(* CoDeSys 2.3.9.50 project: Palettierer.pro *)
(* Libraries: TcIoFunctions.lib 20.1.15 18:06:58, TcXmlDataSrv.lib 11.7.11 07:38:08, STANDARD.LIB 5.6.98 13:03:02, TcBase.lib 14.5.09 13:14:08, TcEtherCAT.lib 9.1.15 17:08:56, TcMath.lib 23.9.04 16:15:30, TcSystem.lib 21.1.15 11:22:54, TcUtilities.lib 6.1.15 17:45:04, TcBaseMath.lib 27.7.04 13:07:56, TcTestAndSet.lib 23.2.09 13:50:08, TcpIp.lib 6.5.15 10:25:52, TcSocketHelper.lib 29.8.14 13:06:24, TcMDP.lib 5.12.13 13:01:38 *)

(* Global variable list: zLibrary/EsponRobot/gEpsonRobot *)
VAR_GLOBAL
	POS_PARK				: DINT := 1;
	POS_RT				: DINT := 21;
	POS_RT_WAIT			: DINT := 22;
	POS_WT_POS1		: DINT := 31;
	POS_WT_POS1_WAIT	: DINT := 32;
	POS_WT_POS2		: DINT := 35;
	POS_CAM_POS1		: DINT := 41;
	POS_CAM_POS2		: DINT := 45;
	POS_NOK				: DINT := 51;
	POS_FEED_PAL_WAIT 	: DINT := 100;
	POS_BUFFER_WAIT	: DINT := 100;
	POS_PAL_WAIT		: DINT := 200;
	POS_TEST_PARTS		: DINT := 300;
END_VAR

(* Global variable list: System/gGlobalSystem *)
VAR_GLOBAL
	Color 					: sColorCode;

	gReadyForControlOn		: BOOL;

	vGlbImpuls_1000ms		: BOOL;
	vGlbImpuls_0500ms		: BOOL;
	vGlbImpuls_0100ms		: BOOL;
	vGlbImpuls_0050ms		: BOOL;
	vGlbImpuls_0025ms		: BOOL;

(*Global Vars for Behr-System-Control *)
	gTipImp					: BOOL;
	gResetAll				: BOOL;
	gInitCollect				: BOOL;
	gInitOk					: BOOL;
	gSetupOk				: BOOL;
	gHomeOk				: BOOL;

(*SystemFlags for SFCs*)
	SFCInit					: BOOL:= FALSE;	(* Systemvariable for stop and reset an SFC *)
											(* Systemvariable zum stoppen und zurücksetzen einer Kette *)
	SFCQuitError			: BOOL:= FALSE;	(* Systemvariable for quitting an SFCError *)
											(* Systemvariable zum Quittieren des SFCErrors *)
	SFCError				: BOOL:= FALSE;	(* Systemvariable for checking Timeout in the step flow chart *)
											(* Systemvariable zur Anzeige eines Schrittkettentimeouts *)
	SFCErrorStep			: STRING:= '';	(* Systemvariable showing step of SFCError in step flow chart *)
											(* Systemvariable zur Anzeige des Schrittes in der der SFCError auftrat *)
	SFCErrorPOU			: STRING:= '';	(* Systemvariable showing Name of the  step flow chart, where SFCError occurs *)
											(* Systemvariable zur Anzeige des Namens der Schrittkette in der der SFCError auftrat *)
	SFCTip  				: BOOL:= FALSE;	(* Systemvariable zum forcen aller Transitionen auf TRUE (! DO NOT USE !) *)
											(* Systemvariable to force all Transitions*)
	SFCTipMode			: BOOL:= FALSE;	(* Systemvariable zum anhalten der AS-Diagramme an den Transitionen *)
											(* Systemvariable to stop an AS-Diagram at the transition *)
	gVarStrSystemTime 		: STRING;
	gVarDTSystemtime		: DT;
	gVarSystemtime			: TIMESTRUCT;

	LocalAmsNetIdArr		: T_AmsNetIdArr;
	LocalAmsNetIdStr		: T_AmsNetId;
	Analyze					: AnalyzeExpression;

	st_Hydra8Data			: struct_Hydra8;
	FbExportHydraString		: Fb_ExportHydraString;

	st_ctrl_in_Empty		: struct_ctrl_in;
	st_ctrl_out_Empty		: struct_ctrl_out;

END_VAR
VAR_GLOBAL CONSTANT
	NO_OF_POS_AXIS		: INT :=3;
	NO_OF_ERRORS		: DINT :=30;
	NO_OF_USERS			: DINT :=50;
	NO_OF_FILES			: DINT :=50;
END_VAR

(* Global variable list: System/gGlobalVisuPersist *)
VAR_GLOBAL
	Visu		 AT %MB1000 : sVisu;
	Service		: sMachParaService;
END_VAR

VAR_GLOBAL RETAIN PERSISTENT
	TD			: sTypeData;
	MP			: sMachPara;
	UD			: sUserList;


	sTDHandler 	: sTDHandler;
	sMPHandler 	: sMPHandler;
	ErrorHistory	: ARRAY[0..500] OF ErrorStruct;

	lastTDActivate	: STRING(255);

	(*Gesamt-Zähler (Reset möglich durch Service*)
	gNOKCount			: DINT;

	(*Gesamt-Zähler (Reset nur möglich durch Administrator*)
	gTotalNOKCount		: DINT;


	PersDaten			: sPersDaten;

END_VAR

(* Global variable list: ept/Global_Checks *)
VAR_GLOBAL
	CheckBounds_ErrCnt 			: DINT := 0;
	CheckByteZeroDiv_ErrCnt 		: DINT := 0;
	CheckDWordZeroDiv_ErrCnt 	: DINT := 0;
	CheckRealZeroDiv_ErrCnt 		: DINT := 0;
	CheckWordZeroDiv_ErrCnt 		: DINT := 0;
	CheckRangeSigned_ErrCnt		: DINT := 0;
	CheckRangeUnsigned_ErrCnt	: DINT := 0;
END_VAR

(* Global variable list: zLibrary/Valve/gValve *)
 VAR_GLOBAL
	gValve		:	sValveGlobalVar;
END_VAR

(* Global variable list: System/MachineParameterFix *)
VAR_GLOBAL

	MP_TDPathLocal			: STRING(255) := 'data\TD\';
	MP_TDPathService		: STRING(255):= 'data\TD\Service\';

	MP_LocalDriveRoot		: STRING(255) := 'data\MP\';

	MP_ExportDrive			: STRING:=	'';

	MP_ExportDrivePathTD	: STRING(255):=  'data\TD';
	MP_ExportDrivePathMP	: STRING(255):=  'data\MP';

	LOG_RDPathLocal			: STRING(255) := 'data\RD\';
	LOG_ExportDrivePathRD	: STRING(255):= 'data\RD';

	MP_TDFileExtension		: STRING(10) := '.XML';
	MP_TDSearchString		: STRING :=  '*.xml';
	MP_MPExportFilename		: STRING := 'MachPara.xml';

	s_PLC_name				: STRING(255);
	s_PLC_path				: STRING(255);
	s_Projekt_path			: STRING(255);

	s_tools_path			: STRING(255):= 'tools\';
	s_ud_path				: STRING(255):= 'data\UD\';

END_VAR

(* Global variable list: Station00/ST00_FBs *)
VAR_GLOBAL
	ST00_40_F1 			: FB_DigIn; (* Vorsicherungen Leistung iO *)
	ST03_210_S1 			: FB_DigIn; (* Not-Aus 1 Anlage ausgelöst *)
	ST08_210_S2 			: FB_DigIn; (* Not-Aus 2 Anlage ausgelöst *)
	ST00_X4_16	 		: FB_DigIn; (* Not-Aus Reserve Anlage ausgelöst *) (*entfällt*)
	ST00_200_A1_A1 		: FB_DigIn; (* Not-Aus iO *)
	ST00_220_S1	 		: FB_DigIn; (* Schutztüre 1 geöffnet *)
	ST00_220_S2			: FB_DigIn; (* Schutztüre 2 geöffnet *)
	ST00_230_S2_E1 		: FB_DigIn; (* Schutztüre 1 geschlossen *)
	ST00_240_S1 			: FB_DigIn; (* Schutztüre 9 geschlossen *)
	ST00_226_S1			: FB_DigIn;(*Hubtüre 1 Schleuse Einlauf STN 8 geschlossen*)
	ST00_226_S2			: FB_DigIn;(*Hubtüre 2 Schleuse Einlauf STN 8 geschlossen*)
	ST00_227_S1			: FB_DigIn;(*Hubtüre 3 Schleuse Auslauf STN 8 geschlossen*)
	ST00_227_S2			: FB_DigIn;(*Hubtüre 4 Schleuse Auslauf STN 8 geschlossen*)
	ST00_229_S1			: FB_DigIn;(*Schutztüre Einlauf Tray STN 8 geschlossen*)
	ST00_230_S1			: FB_DigIn;(*Schutztüre Auslauf Tray STN 8 geschlossen*)
	ST00_231_S1			: FB_DigIn;(*Schutztüre Panel / Rutsche STN 8 geschlossen*)
	ST00_232_S1			: FB_DigIn;(*Schutztüre 8 Auslauf Trays STN 8 geschlossen*)
	ST00_170_Motorschutz	: FB_DigIn;(*Motorschutz in Ordnung*)
	ST00_170_Thermokont	: FB_DigIn;(*Thermokontakt in Ordnung*)
	ST00_228_S1			: FB_DigIn;(*Bandstecke EPT angebaut*)
	ST00_71_X1_3  		: FB_DigIn; (* Schnittstelle Bedrucken Tinte JSK auf Übergabeposition *)
	ST00_71_X1_4  		: FB_DigIn; (* Schnittstelle Bedrucken Tinte Druckstation betriebsbereit *)
	ST00_72_X1_3  		: FB_DigIn; (* Schnittstelle Tampondrucker Teil in Abholposition *)(*Band Entnahmeposition 1*)
	ST00_72_X1_8  		: FB_DigIn; (* Schnittstelle Tampondrucker Druck abgeschlossen *)	(*gleich wie ST02_S2_B11_0*)
	ST00_292_S1_STOP 	: FB_DigIn; (* Bedienstelle Produktion Stop *)
	ST00_292_S2_START	: FB_DigIn; (* Bedienstelle Produktion Start *)
	ST00_292_S3_RESET	: FB_DigIn; (* Bedienstelle Produktion Reset *)
	ST00_350_B20_0 		: FB_DigIn; (* Druckschalter Wartungseinheit Hauptluft min.6 bar *)

	ST00_245_V1			: FB_DigOutIn; (* Verriegelung Schutztüren-Leuchte *)
	ST00_245_V2_START	: FB_DigOutIn; (* Bedienstelle Start-Leuchte *)
	ST00_245_V3_RESET	: FB_DigOutIn; (* Bedienstelle Reset-Schutztüren-Leuchte *)
	ST00_245_S1_STOP 	: FB_DigIn;	(* Bedienstelle Produktion Stop *)
	ST00_245_S2_START	: FB_DigIn; (* Bedienstelle Produktion Start *)
	ST00_245_S3_RESET	: FB_DigIn; (* Bedienstelle Produktion Reset *)

	ST00_31_K1 			: FB_DigOutIn; (* Beleuchtung Anlage *)
	ST00_350_H1			: FB_DigOutIn; (* Signalsäule RD Maschine Alarm/Störung *)
	ST00_350_H2			: FB_DigOutIn; (* Signalsäule YE Bedienereingriff erforderlich *)
	ST00_350_H3			: FB_DigOutIn; (* Signalsäule GN Maschine Automatik *)
	ST00_200_A1_E4 		: FB_DigOutIn; (* Quittierung Not-Aus *)
	ST00_220_S1_S31		: FB_DigOutIn; (* Verriegelung Schutztüren *)
	ST00_292_H2_START	: FB_DigOutIn; (* Bedienstelle Start-Leuchte *)
	ST00_292_H3_RESET	: FB_DigOutIn; (* Bedienstelle Reset-Leuchte *)

	ST00_71_K2	  		: FB_DigOutIn; (* Schnittstelle Bedrucken Tinte Abholposition frei *)
	ST00_72_K7	  		: FB_DigOutIn; (* Schnittstelle Tampondrucker Reset  Rundtisch *)

	ST00_73_K3	  		: FB_DigOutIn; (* Schnittstelle Förderband frei für Spritzmaschine*)
	ST00_73_K4	  		: FB_DigIn; 		(* Schnittstelle Freigabe von Spritzmaschine (nur für Anlagen ohne Rundtisch)*)
	ST00_74_B7_2    		: FB_ValveSensor; (* Stopper GST1 DS*)
	ST00_74_B7_3   		: FB_ValveSensor; (* Stopper GST2 PS*)
	ST00_74_B7_4    		: FB_ValveSensor; (* Vereinzeler AST1 DS*)
	ST00_74_B7_5   	 	: FB_ValveSensor; (* Vereinzeler AST2 PS*)
	ST00_74_B7_6  	 	: FB_ValveSensor; (* Vereinzeler GST1 DS*)
	ST00_74_B7_7   		: FB_ValveSensor; (* Vereinzeler GST2 PS*)

	ST00_74_Y2_4    		: FB_Valve; (*ST00_74_Y2_4 Stopper Bandstrecke (Valve) *)
	ST00_74_Y2_5    		: FB_Valve; (*ST00_74_Y2_5 Vereinzeler Bandstrecke (Valve) *)

END_VAR

(* Global variable list: Station00/ST00_Global *)
VAR_GLOBAL
	gDisableMP				: BOOL := FALSE;		(* deaktivieren der Maschinenparamtereingabe *)
	gDisableTD				: BOOL := FALSE;		(* deaktivieren der Typedateneingabe *)

	gHomePosSFCDone		: BOOL;
	gResetButton		: BOOL;
	gRobotOffset		: DINT;
	gTypeCode		  	: DINT;
	ProcessMessage01	: STRING(80);
	ProcessMessage02	: STRING(80);
	gTInfo_FirstStart	: BOOL;
	gBasicManualMode	: BOOL;
	SpecialModeProgNu	: DINT;

	gStartRunEmpty		: BOOL;
	gRunEmpty			: BOOL;

	DummyTest_160pol	: BOOL;
	Dummy_test_Result	: ARRAY[1..MAX_NO_OF_DUMMYS] OF BOOL;
	Dummy_test_Vorgabe	: ARRAY[1..MAX_NO_OF_DUMMYS] OF BOOL;

END_VAR
VAR_GLOBAL RETAIN PERSISTENT
	gTypeDataValid		 : BOOL;
END_VAR
VAR_GLOBAL CONSTANT
	MAX_NO_OF_DUMMYS	: DINT := 6;
END_VAR

(* Global variable list: Station00/ST00_VarVonfig *)
VAR_CONFIG
	BusDiagnosis.EtheCatMasterAmsNetId AT %IB1000 : ARRAY [0..5] OF USINT;

(* Vorsicherungen Leistung iO *)
.ST00_40_F1.BitInToCheck                 	AT %IX0.0 : BOOL;
(* Schutztüre 2 geöffnet *)
.ST00_220_S2.BitInToCheck                 AT %IX0.2 : BOOL;
(* Not-Aus 1 Anlage ausgelöst *)
.ST03_210_S1.BitInToCheck                 AT %IX0.3 : BOOL;
(* Not-Aus 2 Anlage ausgelöst *)
.ST08_210_S2.BitInToCheck                 AT %IX0.4 : BOOL;
(* Not-Aus Reserve Anlage ausgelöst *)
.ST00_X4_16.BitInToCheck                 	AT %IX0.5 : BOOL;
(* Not-Aus iO *)
.ST00_200_A1_A1.BitInToCheck              AT %IX0.6 : BOOL;
(* Schutztüre 9 geschlossen *)
.ST00_240_S1.BitInToCheck                 AT %IX0.7 : BOOL;
(* Schutztüre 1 geöffnet *)
.ST00_220_S1.BitInToCheck                 AT %IX1.0 : BOOL;
(* Schutztüre 1 geschlossen *)
.ST00_230_S2_E1.BitInToCheck              AT %IX1.1 : BOOL;
(*Hubtüre 1 Schleuse Einlauf STN 8 geschlossen*)
.ST00_226_S1.BitInToCheck                 AT %IX1.2 : BOOL;
(*Hubtüre 2 Schleuse Einlauf STN 8 geschlossen*)
.ST00_226_S2.BitInToCheck                 AT %IX1.3 : BOOL;
(*Hubtüre 3 Schleuse Auslauf STN 8 geschlossen*)
.ST00_227_S1.BitInToCheck                 AT %IX1.4 : BOOL;
(*Hubtüre 4 Schleuse Auslauf STN 8 geschlossen*)
.ST00_227_S2.BitInToCheck                 AT %IX1.5 : BOOL;
(*Motorschutz in Ordnung*)
	ST00_170_Motorschutz.BitInToCheck	AT %IX1.6 : BOOL;
(*Thermokontakt in Ordnung*)
	ST00_170_Thermokont.BitInToCheck	AT %IX1.7 : BOOL;

(* Schnittstelle Bedrucken Tinte JSK auf Übergabeposition *)
.ST00_71_X1_3.BitInToCheck                AT %IX2.0 : BOOL;
(* Schnittstelle Bedrucken Tinte Druckstation betriebsbereit *)
.ST00_71_X1_4.BitInToCheck                AT %IX2.1 : BOOL;
(* Schnittstelle Tampondrucker Teil in Abholposition *)
.ST00_72_X1_3.BitInToCheck                AT %IX2.2 : BOOL;

(* Schnittstelle Tampondrucker Druck abgeschlossen *)
.ST00_72_X1_8.BitInToCheck                AT %IX2.7 : BOOL;
(*Bandstecke EPT angebaut*)
.ST00_228_S1.BitInToCheck                 AT %IX3.0 : BOOL;

(*Schutztüre Einlauf Tray STN 8 geschlossen*)
.ST00_229_S1.BitInToCheck                 AT %IX3.2 : BOOL;
(*Schutztüre Auslauf Tray STN 8 geschlossen*)
.ST00_230_S1.BitInToCheck                 AT %IX3.3 : BOOL;
(*Schutztüre Panel / Rutsche STN 8 geschlossen*)
.ST00_231_S1.BitInToCheck                 AT %IX13.0 : BOOL;
(*Schutztüre 8 Auslauf Trays STN 8 geschlossen*)
.ST00_232_S1.BitInToCheck                 AT %IX13.1 : BOOL;

(* Bedienstelle Produktion Stop *)
.ST00_292_S1_STOP.BitInToCheck            AT %IX3.5 : BOOL;
(* Bedienstelle Produktion Start *)
.ST00_292_S2_START.BitInToCheck           AT %IX3.6 : BOOL;
(* Bedienstelle Produktion Start *)
.ST00_292_S3_RESET.BitInToCheck           AT %IX3.7 : BOOL;
(* Druckschalter Wartungseinheit Hauptluft min.6 bar *)
.ST00_350_B20_0.BitInToCheck           		AT %IX20.0 : BOOL;

(* Beleuchtung Anlage *)
.ST00_31_K1.BitInToCheck             		: BOOL := FALSE;
.ST00_31_K1.BitOutToSet              		  AT %QX0.0 : BOOL;
(* Signalsäule RD Maschine Alarm/Störung *)
.ST00_350_H1.BitInToCheck             	: BOOL := FALSE;
.ST00_350_H1.BitOutToSet              	  AT %QX0.4 : BOOL;
(* Signalsäule YE Bedienereingriff erforderlich *)
.ST00_350_H2.BitInToCheck             	: BOOL := FALSE;
.ST00_350_H2.BitOutToSet              	  AT %QX0.5 : BOOL;
(* Signalsäule GN Maschine Automatik *)
.ST00_350_H3.BitInToCheck             	: BOOL := FALSE;
.ST00_350_H3.BitOutToSet              	  AT %QX0.6 : BOOL;
(* Quittierung Not-Aus *)
.ST00_200_A1_E4.BitInToCheck            : BOOL := FALSE;
.ST00_200_A1_E4.BitOutToSet               AT %QX1.0 : BOOL;
(* Verriegelung Schutztüren *)
.ST00_220_S1_S31.BitInToCheck           : BOOL := FALSE;
.ST00_220_S1_S31.BitOutToSet              AT %QX1.1 : BOOL;
(* Bedienstelle Start-Leuchte *)
.ST00_292_H2_START.BitInToCheck         : BOOL := FALSE;
.ST00_292_H2_START.BitOutToSet            AT %QX1.5 : BOOL;
(* Bedienstelle Reset-Leuchte *)
.ST00_292_H3_RESET.BitInToCheck         : BOOL := FALSE;
.ST00_292_H3_RESET.BitOutToSet            AT %QX1.7 : BOOL;

(* Schnittstelle Bedrucken Tinte Abholposition frei *)
.ST00_71_K2.BitInToCheck             		: BOOL := FALSE;
.ST00_71_K2.BitOutToSet              		  AT %QX2.1 : BOOL;

(* Schnittstelle Förderband frei für Spritzmaschine*)
.ST00_73_K3.BitInToCheck             		: BOOL := FALSE;
.ST00_73_K3.BitOutToSet              		  AT %QX0.7 : BOOL;


(*ST00_74_Y2_4 Stopper Bandstrecke (Valve) *)
.ST00_74_Y2_4.CoilA                    AT %QX2.4 : BOOL;
.ST00_74_Y2_4.CoilB                    AT %MX2.4 : BOOL;

(*ST00_74_Y2_5 Vereinzeler Bandstrecke (Valve) *)
.ST00_74_Y2_5.CoilA                    AT %QX2.5 : BOOL;
.ST00_74_Y2_5.CoilB                    AT %MX2.5 : BOOL;

(*ST00_74_B7_2 Stopper GST1 DS (DigIn) *)
.ST00_74_B7_2.ValveSensor             AT %IX7.2 : BOOL;

(*ST00_74_B7_3 Stopper GST2 PS (DigIn) *)
.ST00_74_B7_3.ValveSensor             AT %IX7.3 : BOOL;

(*ST00_74_B7_4 Vereinzeler AST1 DS (DigIn) *)
.ST00_74_B7_4.ValveSensor             AT %IX7.4 : BOOL;

(*ST00_74_B7_5 Vereinzeler AST2 PS (DigIn) *)
.ST00_74_B7_5.ValveSensor             AT %IX7.5 : BOOL;

(*ST00_74_B7_6 Vereinzeler GST1 DS (DigIn) *)
.ST00_74_B7_6.ValveSensor          AT %IX7.6: BOOL;

(*ST00_74_B7_7 Vereinzeler GST2 PS(DigIn) *)
.ST00_74_B7_7.ValveSensor             AT %IX7.7 : BOOL;


END_VAR

(* Global variable list: Station02/ST02_FBs *)
VAR_GLOBAL
	ST02_FDB_55X1_5_READY		:FB_DigIn; (* IFM Kamera Flügelerkennung links Ready *)
	ST02_FDB_55X1_6_IO			 :FB_DigIn; (* IFM Kamera Flügelerkennung links Ergebnis iO *)
	ST02_FDB_55X1_6_NIO		:FB_DigIn; (* IFM Kamera Flügelerkennung links Ergebnis niO *)
	ST02_FDB_55X1_2_TRIGGER	:FB_DigOutIn; (* IFM Kamera Flügelerkennung links Trigger *)
	ST02_FDB_55X1_7_JOB_BIT1 	:FB_DigOutIn; (* IFM Kamera links  Jobwechsel Bit 1 *)
	ST02_FDB_55X1_7_JOB_BIT2 	:FB_DigOutIn; (* IFM Kamera links Jobwechsel Bit 2 *)

	ST02_FDB_56X1_5_READY		:FB_DigIn; (* IFM Kamera Flügelerkennung rechts Ready *)
	ST02_FDB_56X1_6_IO			:FB_DigIn; (* IFM Kamera Flügelerkennung rechts Ergebnis iO *)
	ST02_FDB_56X1_6_NIO		:FB_DigIn; (* IFM Kamera Flügelerkennung rechts Ergebnis niO *)
	ST02_FDB_56X1_2_TRIGGER	:FB_DigOutIn; (* IFM Kamera Flügelerkennung rechts Trigger *)
	ST02_FDB_56X1_7_JOB_BIT1	:FB_DigOutIn; (* IFM Kamera links  Jobwechsel Bit 1 *)
	ST02_FDB_56X1_7_JOB_BIT2	:FB_DigOutIn; (* IFM Kamera links Jobwechsel Bit 2 *)


	ST02_DT_95_A1 			:FB_Sensopart;	(*Sensopart Kamera Farberkennung*)
	ST02_DT_95_A2 			:FB_SensopartEthernet;	(*Sensopart Kamera Farberkennung*)

	ST02_S1_70K61_A1		:FB_DigOutIn; 	(* Start  Bedrucken *)

	ST02_DT_62_B11		:FB_ValveSensor;	(* Schwenkarm 1 0 Grad*)
	ST02_DT_61_B21		:FB_ValveSensor;	(* Schwenkarm 2 90 Grad*)
	ST02_DT_61_B11		:FB_ValveSensor;	(* Schwenkarm 2 180 Grad*)
	ST02_DT_61_B31		:FB_ValveSensor;	(* Schwenkarm 2 0 Grad*)
	ST02_DT_61_B41 		:FB_ValveSensor;	(* Schwenkarm 1 180 Grad*)
	ST02_DT_61_B51 		:FB_ValveSensor;	(* Schwenkarm 1 90 Grad*)
	ST02_FDB_54_B11		:FB_ValveSensor; 	(* Kamera Ausschleusen Bandstrecke eingefahren GST*)
	ST02_FDB_54_B21		:FB_ValveSensor; 	(* Kamera Ausschleusen Bandstrecke ausgefahren AST*)
	ST02_S1_66_B11 		:FB_ValveSensor;	(*9: Schwenkarm 1 ISK Fixierung GST*)
	ST02_S1_66_B21 		:FB_ValveSensor;	(*10: Schwenkarm 1 ISK Fixierung AST*)
	ST02_S1_66_B31 		:FB_ValveSensor;	(*11: Schwenkarm 2 ISK Fixierung GST*)
	ST02_S1_66_B41	 	:FB_ValveSensor;	(*12: Schwenkarm 2 ISK Fixierung AST*)

	ST02_FDB_40_B61		:FB_DigIn; (* Iso von SPM auf Band abgelegt *)
	ST02_FDB_40_B71		:FB_DigIn; (* Iso auf Band vor Vereinzler *)

	ST02_DT_62_B81		:FB_ValveSensor; 	(* Tisch drehen 0 Grad*)			(*gleich wie ST00_72_X1_6*)
	ST02_DT_62_B91		:FB_ValveSensor;	(* Tisch drehen 180 Grad*)			(*gleich wie ST00_72_X1_7*)
	ST02_S1_40K01 		:FB_DigIn;			(* Freigabe Förderband von SPM*)

	ST02_FDB_80_B02 		:FB_DigIn;			(* Band Entnahmeposition 2 102pol*)
	ST02_FDB_54_B41		:FB_DigIn; 			(* Kamera ISK anwesend an Prüfposition nur zum Schlechtteile zählen*)
	ST02_35_S31 			:FB_DigIn; 			(* ST02 Druckschalter Wartungseinheit Hauptluft min.6 bar *)
	ST02_S1_6A01			:FB_DigIn; 			(* ST02 Sicherung 24V *)

	ST02_35Y01			:FB_Valve; 			(*1: Einschaltventil Hauptluft Tampondruckanlage*)

	ST02_62_Y4  			:FB_Valve; 			(*Kamera Ausschleusen Bandstrecke (Valve) *)
	ST02_62_Y6			:FB_Valve; 			(*Tisch drehen 0 - 180 Grad (Valve) *)

	ST02_Schwenkarm	: ARRAY[1..2] OF FB_Schwenken;
	ST02_62_Y9			:FB_Valve; 			(*Schwenkarm 2 drehen 90 - 180 Grad (Valve) *)
	ST02_62_Y11			:FB_Valve; 			(*Schwenkarm 2 drehen 90 - 0 Grad (Valve) *)

	ST02_62_Y13			:FB_Valve; 			(*Schwenkarm 1 drehen 90 - 180 Grad (Valve) *)
	ST02_62_Y15			:FB_Valve; 			(*Schwenkarm 1 drehen 90 - 0 Grad (Valve) *)

	ST02_62_Y17			:FB_Valve; 			(*Schwenkarm 1 ISK Fixierung ein/ausfahren(Valve)*)
	ST02_62_Y18			:FB_Valve; 			(*Schwenkarm 2 ISK Fixierung ein/ausfahren(Valve)*)

	ST02_DT_65B11  		:FB_DigIn;			(* Tampondrucker Nest 1 leer *)
	ST02_DT_65B21		:FB_DigIn; 			(* Tampondrucker Nest 2 leer *)

END_VAR

(* Global variable list: Station02/ST02_Global *)
VAR_GLOBAL
	gTableEmpty			: BOOL;
END_VAR

VAR_GLOBAL CONSTANT
	NO_OF_NEST			: INT := 2;		(* No of Nests on TurnTable *)
END_VAR

(* Global variable list: Station02/ST02_VarVonfig *)
(* Generated automatically by TwinCAT - (read only) *)
VAR_CONFIG

(*ST02_FDB_55X1_5_READY IFM Kamera Flügelerkennung links Ready (DigIn) *)
.ST02_FDB_55X1_5_READY.BitInToCheck           AT %IX100.1 : BOOL;
(*ST02_FDB_55X1_6_IO IFM Kamera Flügelerkennung links Ergebnis iO (DigIn) *)
.ST02_FDB_55X1_6_IO.BitInToCheck         		  AT %IX100.2 : BOOL;
(*ST02_FDB_55X1_6_NIO IFM Kamera Flügelerkennung links Ergebnis niO (DigIn) *)
.ST02_FDB_55X1_6_NIO.BitInToCheck        		   AT %IX100.3 : BOOL;
(*ST02_FDB_55X1_2_TRIGGER IFM Kamera Flügelerkennung links Trigger (DigOutIn) *)
.ST02_FDB_55X1_2_TRIGGER.BitInToCheck                : BOOL := FALSE;
.ST02_FDB_55X1_2_TRIGGER.BitOutToSet                 AT %QX100.1 : BOOL;
(* IFM Kamera links  Jobwechsel Bit 1 *)
.ST02_FDB_55X1_7_JOB_BIT1.BitInToCheck                : BOOL := FALSE;
.ST02_FDB_55X1_7_JOB_BIT1.BitOutToSet                 AT %QX100.2 : BOOL;
(* IFM Kamera links Jobwechsel Bit 2 *)
.ST02_FDB_55X1_7_JOB_BIT2.BitInToCheck                : BOOL := FALSE;
.ST02_FDB_55X1_7_JOB_BIT2.BitOutToSet                 AT %QX100.3 : BOOL;

(*ST02_FDB_56X1_5_READY IFM Kamera Flügelerkennung rechts Ready (DigIn) *)
.ST02_FDB_56X1_5_READY.BitInToCheck           AT %IX101.4 : BOOL;
(*ST02_FDB_56X1_6_IO IFM Kamera Flügelerkennung rechts Ergebnis iO (DigIn) *)
.ST02_FDB_56X1_6_IO.BitInToCheck           AT %IX101.5 : BOOL;
(*ST02_FDB_56X1_6_NIO IFM Kamera Flügelerkennung rechts Ergebnis niO (DigIn) *)
.ST02_FDB_56X1_6_NIO.BitInToCheck           AT %IX101.6 : BOOL;
(*ST02_FDB_56X1_2_TRIGGER IFM Kamera Flügelerkennung rechts Trigger (DigOutIn) *)
.ST02_FDB_56X1_2_TRIGGER.BitInToCheck                : BOOL := FALSE;
.ST02_FDB_56X1_2_TRIGGER.BitOutToSet                 AT %QX101.2 : BOOL;
(* IFM Kamera rechts  Jobwechsel Bit 1 *)
.ST02_FDB_56X1_7_JOB_BIT1.BitInToCheck                : BOOL := FALSE;
.ST02_FDB_56X1_7_JOB_BIT1.BitOutToSet                 AT %QX101.3 : BOOL;
(* IFM Kamera rechts Jobwechsel Bit 2 *)
.ST02_FDB_56X1_7_JOB_BIT2.BitInToCheck                : BOOL := FALSE;
.ST02_FDB_56X1_7_JOB_BIT2.BitOutToSet                 AT %QX101.4 : BOOL;


(*ST02_S1_70K61_A1 Start  Bedrucken (DigOutIn) *)
.ST02_S1_70K61_A1.BitInToCheck                : BOOL := FALSE;
.ST02_S1_70K61_A1.BitOutToSet                 AT %QX6.3: BOOL;

(*ST02_S1_40K01 Freigabe Förderband von SPM (DigIn)*)
.ST02_S1_40K01.BitInToCheck    AT %IX11.2 : BOOL;
(*ST02_FDB_80_B02  Band Entnahmeposition 2(DigIn) *)
.ST02_FDB_80_B02.BitInToCheck    AT %IX11.6 : BOOL;

(* Tampondrucker Nest 1 leer *)
.ST02_DT_65B11.BitInToCheck                AT %IX2.3 : BOOL;
(* Tampondrucker Nest 2 leer *)
.ST02_DT_65B21.BitInToCheck                AT %IX2.4 : BOOL;

(*ST02_DT_62_B11 Schwenkarm 1 0 Grad (DigIn) *)
.ST02_DT_62_B11.ValveSensor             AT %IX10.0 : BOOL;
(*ST02_DT_61_B21 Schwenkarm 2 90 Grad(DigIn) *)
.ST02_DT_61_B21.ValveSensor             AT %IX10.1 : BOOL;
(*ST02_DT_61_B11 Schwenkarm 2 180 Grad(DigIn) *)
.ST02_DT_61_B11.ValveSensor             AT %IX10.2 : BOOL;
(*ST02_DT_61_B31 Schwenkarm 2 0 Grad(DigIn) *)
.ST02_DT_61_B31.ValveSensor             AT %IX10.3 : BOOL;
(*ST02_DT_61_B41 Schwenkarm 1 180 Grad(DigIn) *)
.ST02_DT_61_B41.ValveSensor             AT %IX10.4 : BOOL;
(*ST02_DT_61_B51 Schwenkarm 1 90 Grad(DigIn) *)
.ST02_DT_61_B51.ValveSensor             AT %IX10.5 : BOOL;
(*ST02_DT_62_B81 Tisch drehen 0 Grad(DigIn) *)
.ST02_DT_62_B81.ValveSensor             AT %IX10.6 : BOOL;
(*ST02_DT_62_B91 Tisch drehen 180 Grad(DigIn) *)
.ST02_DT_62_B91.ValveSensor             AT %IX10.7 : BOOL;
(*
(*ST02_S1_66_B11 Schwenkarm 1 ISK Fixierung GST(DigIn) *)
.ST02_S1_66_B11.ValveSensor             AT %I* : BOOL;
(*ST02_S1_66_B21 Schwenkarm 1 ISK Fixierung AST(DigIn) *)
.ST02_S1_66_B21.ValveSensor             AT %I* : BOOL;
(*ST02_S1_66_B31 Schwenkarm 2 ISK Fixierung GST(DigIn) *)
.ST02_S1_66_B31.ValveSensor             AT %I* : BOOL;
(*ST02_S1_66_B41 Schwenkarm 2 ISK Fixierung AST(DigIn) *)
.ST02_S1_66_B41.ValveSensor             AT %I* : BOOL;

(* ST02 Druckschalter Wartungseinheit Hauptluft min.6 bar *)
.ST02_35_S31.BitInToCheck             AT %I* : BOOL;
(* ST02 Sicherung 24V *)
.ST02_S1_6A01.BitInToCheck             AT %I* : BOOL;
*)
(*
(*ST02_62V9a Schwenkarm 1 ISK Fixierung ein/ausfahren(Valve) (Valve) *)
.ST02_62V9a.CoilA                    AT %Q* : BOOL;
(*ST02_62V9b Schwenkarm 2 ISK Fixierung ein/ausfahren(Valve)  (Valve) *)
.ST02_62V9b.CoilB                    AT %Q* : BOOL;
*)
(*
(*ST02_62_Y6 Tisch drehen 0 - 180 Grad  (Valve) *)
.ST02_62_Y6.CoilA                    AT %QX5.6 : BOOL;
.ST02_62_Y6.CoilB                    AT %MX5.6 : BOOL;
(*ST02_62_Y9 Schwenkarm 2 drehen 90 - 180 Grad  (Valve) *)
.ST02_62_Y9.CoilA                    AT %QX5.7 : BOOL;
.ST02_62_Y9.CoilB                    AT %MX5.7 : BOOL;
(*ST02_62_Y11 Schwenkarm 2 drehen 90 - 0 Grad  (Valve) *)
.ST02_62_Y11.CoilA                    AT %QX6.0 : BOOL;
.ST02_62_Y11.CoilB                    AT %MX6.0 : BOOL;
(*ST02_62_Y13 Schwenkarm 1 drehen 90 - 180 Grad  (Valve) *)
.ST02_62_Y13.CoilA                    AT %QX6.1 : BOOL;
.ST02_62_Y13.CoilB                    AT %MX6.1 : BOOL;
(*ST02_62_Y15 Schwenkarm 1 drehen 90 - 0 Grad  (Valve) *)
.ST02_62_Y15.CoilA                    AT %QX6.2 : BOOL;
.ST02_62_Y15.CoilB                    AT %MX6.2 : BOOL;
*)
(*ST02_62_Y4 Kamera Ausschleusen Bandstrecke (Valve) *)
.ST02_62_Y4.CoilA                    AT %QX60.0 : BOOL;
.ST02_62_Y4.CoilB                    AT %QX60.1 : BOOL;

(*ST02_FDB_54_B11 Kamera Ausschleusen Bandstrecke eingefahren (DigIn) *)
.ST02_FDB_54_B11.ValveSensor             AT %IX60.0 : BOOL;
(*ST02_FDB_54_B21 Kamera Ausschleusen Bandstrecke ausgefahren (DigIn) *)
.ST02_FDB_54_B21.ValveSensor             AT %IX60.1 : BOOL;

(*ST02_FDB_54_B41 Kamera ISK anwesend an Prüfposition (DigIn) *)
.ST02_FDB_54_B41.BitInToCheck           AT %IX70.6 : BOOL;
(*
(*ST02_35Y01 Einschaltventil Hauptluft Tampondruckanlage (Valve) *)
.ST02_35Y01.CoilA                    AT %Q* : BOOL;
.ST02_35Y01.CoilB                    AT %Q* : BOOL;*)
END_VAR

(* Global variable list: Station03/ST03_FBs *)
VAR_GLOBAL

	ST03_51_M1	: fb_72x1_Achse;	(* Förderbandmotor*)
	ST03_601V1_A1: FB_DigOutIn;		(* Förderband Prüfteile *)
	ST03_A5		: FB_DigOutIn;		(* Förderbandmotor Oriental *)
	ST03_V2	 	: FB_DigIn; 		(* Störung Motor Förderband Oriental *)

	ST03_125_F1 : FB_DigIn; 		(* Absicherung Roboter iO *)
	Robot01		: FB_EpsonRobot;

	St03_120_A1_A14: FB_DigIn;		(* Roboter opt.- Tool 2 ist ein*)
	ST03_400_B12_6 : FB_DigIn; 		(* Schwenkmodul AST (Roboterkopf) *)
	ST03_400_B12_7 : FB_DigIn; 		(* Schwenkmodul GST (Roboterkopf) *)
	ST03_400_B54_7: FB_DigIn; 		(* Tray Testteile in Position *)
	ST03_8_75_B13_5: FB_DigIn; 		(* voll/belegt keine Prüfmittel mehr*)
	ST03_8_75_B13_6: FB_DigIn; 		(* belegt mit 6 Prüfmitteln*)

	ST03_BG3_S53_0:FB_DigIn;		(* Start Band für Dummyprüfung*)
	ST03_BG3_X53_0:	FB_DigOutIn;	(* LED TasterStart Band für Dummyprüfung*)

	ST03_65_Q1: FB_DigOutIn;		(* Kühltunnel (Lüfter)*)
	ST03_65_F1: FB_DigIn;			(* Sicherung Kühltunnel (Lüfter)*)

	ST03_8_100_A1	: FB_SensopartEthernet;	(*Sensopart Kamera Farberkennung*)
	ST03_8_103_A1	: FB_SensopartEthernet;	(*Sensopart Kamera Farberkennung*)

	(*Rüstsatz 154 Rasterplatte======================================================================================*)
	ST03_418_B60_0: FB_ValveSensor; (* Förderband linke Zuführung Vereinzler AST*)
	ST03_418_B60_1: FB_ValveSensor; (* Förderband linke Zuführung Vereinzler GST*)
	ST03_418_B60_2: FB_ValveSensor; (* Förderband rechte Zuführung Vereinzler AST*)
	ST03_418_B60_3: FB_ValveSensor; (* Förderband rechte Zuführung Vereinzler GST*)
	ST03_418_B60_4: FB_ValveSensor; (* Förderband links/rechts Zuführung Stopper AST*)
	ST03_418_B60_5: FB_ValveSensor;	(* Förderband links/rechts Zuführung Stopper GST*)

	ST03_418_B60_6: FB_DigIn;		(* Zuführung links frei zum Ablegen ISK SP Maschine *)
	ST03_418_B60_7: FB_DigIn;		(* Zuführung rechts frei zum Ablegen ISK SP Maschine *)

	ST03_419_B61_0: FB_DigIn;		(* Förderband Zuführung links ISK anwesend zum Vereinzeln*)
	ST03_419_B61_1: FB_DigIn;		(* Förderband Zuführung rechts ISK anwesend zum Vereinzeln*)
	ST03_419_B61_2: FB_DigIn;		(* Züführung links ISK auf Übergabeposition Roboter Palettierer*)
	ST03_419_B61_3: FB_DigIn;		(* Züführung rechts ISK auf Übergabeposition Roboter Palettierer*)

	ST03_419_Y61_5 : FB_Valve; 		(* Förderband linke Zuführung Vereinzler AST/GST *)
	ST03_419_Y61_6 : FB_Valve; 		(* Förderband rechte Zuführung Vereinzler AST/GST *)
	ST03_419_Y61_7 : FB_Valve; 		(* Förderband links/rechts Züführung Stopper AST/GST *)

	(*Rüstsatz 154 pol======================================================================================*)
	ST03_425_B67_0: FB_ValveSensor; (* Förderbandeinheit  Zuführung Vereinzler AST*)
	ST03_425_B67_1: FB_ValveSensor; (* Förderbandeinheit  Zuführung Vereinzler GST*)
	ST03_425_B67_2: FB_ValveSensor; (* Förderbandeinheit  Zuführung Stopper AST*)
	ST03_425_B67_3: FB_ValveSensor; (* Förderbandeinheit  Zuführung Stopper GST*)
	ST03_425_B67_4: FB_DigIn;		(* Zuführung  frei zum Ablegen ISK SP Maschine Pos.1 *)
	ST03_425_B67_5: FB_DigIn;		(* Zuführung  frei zum Ablegen ISK SP Maschine Pos.2 *)
	ST03_425_B67_6: FB_DigIn;		(* Zuführung  frei zum Ablegen ISK SP Maschine Pos.3 *)
	ST03_425_B67_7: FB_DigIn;		(* ISK anwesend am Vereinzler*)

	ST03_426_B68_4: FB_DigIn;		(* Züführung  ISK auf Übergabeposition Roboter Palettierer*)
	ST03_426_Y68_5 : FB_Valve; 		(* Förderband  Zuführung Vereinzler AST/GST *)
	ST03_426_Y68_6 : FB_Valve; 		(* Förderband  Züführung Stopper AST/GST *)

	(*Rüstsatz 160pol======================================================================================*)
	ST03_421_B63_0: FB_ValveSensor; (* Förderband Zuführung Vereinzler AST*)
	ST03_421_B63_1: FB_ValveSensor; (* Förderband Zuführung Vereinzler GST*)
	ST03_421_B63_2: FB_ValveSensor;	(* Förderband Zuführung Stopper AST*)
	ST03_421_B63_3: FB_ValveSensor; (* Förderband Zuführung Stopper GST*)
	ST03_421_B63_4: FB_DigIn;		(* Förderband frei zum Ablegen ISK SP Maschine Pos1 *)
	ST03_421_B63_5: FB_DigIn;		(* Förderband frei zum Ablegen ISK SP Maschine Pos2 *)
	ST03_421_B63_6: FB_DigIn;		(* Förderband frei zum Ablegen ISK SP Maschine Pos3 *)
	ST03_421_B63_7: FB_DigIn;		(* ISK anwesend am Vereinzler*)

	ST03_422_B64_0: FB_DigIn;		(* Förderband Trigger Tintenstrahldrucker 1 (Lichtschranke) Rüstsatz*)
	ST03_423_B66_0: FB_DigIn;		(* Förderband Trigger Tintenstrahldrucker 2 (Lichtschranke) Rüstsatz*)
	ST03_8_B76_1: FB_DigIn;			(* Förderband Trigger Tintenstrahldrucker 1 (Lichtschranke) 3621 *)
	ST03_8_B76_2: FB_DigIn;			(* Förderband Trigger Tintenstrahldrucker 2 (Lichtschranke) 3621 *)
	ST03_422_B64_1: FB_ValveSensor;	(* Förderband Zuführung Stopper 1 Kamera AST*)
	ST03_422_B64_2: FB_ValveSensor; (* Förderband Zuführung Stopper 1 Kamera GST*)
	ST03_422_B64_3: FB_DigIn;		(* Förderband ISK anwesend Stopper 1 Kamera*)
	ST03_422_B64_4: FB_DigIn; 		(* Zuführung ISK auf Übergabeposition Robo Palettierer*)

	ST03_422_Y64_5 : FB_Valve; 		(* Förderband  Zuführung Vereinzler AST/GST *)
	ST03_422_Y64_6 : FB_Valve; 		(* Förderband  Stopper Vereinzler AST/GST *)
	ST03_422_Y64_7 : FB_Valve; 		(* Förderband  Stopper 1 Kamera AST/GST *)

	ST03_423_B65_0: FB_ValveSensor;	(* Förderband Zuführung Stopper 2 Kamera AST*)
	ST03_423_B65_1: FB_ValveSensor;	(* Förderband Zuführung Stopper 2  Kamera GST*)
	ST03_423_B65_2: FB_DigIn; 		(* Förderband ISK anwesend Stopper 2 Kamera*)
	ST03_423_B65_3: FB_ValveSensor;	(* Förderband Zuführung Stopper 3 Kamera AST*)
	ST03_423_B65_4: FB_ValveSensor; (* Förderband Zuführung Stopper 3 Kamera GST*)
	ST03_423_B65_5: FB_DigIn;		(* Förderband ISK anwesend Stopper 3 Kamera*)

	ST03_423_Y65_6 : FB_Valve; 		(* Förderband  Stopper 2 Kamera AST/GST *)
	ST03_423_Y65_7 : FB_Valve; 		(* Förderband  Stopper 3 Kamera AST/GST *)

	ST03_33F4: FB_DigIn; 	(*Steckdosen Tintenstrahldrucker*)				(*212_A14  I1*)
	ST03_70U3_1: FB_DigIn; 	(*Bereit/ Im Druck Tintenstrahldrucker Frontseite*)	(*212_A14  I2*)
	ST03_70U3_2: FB_DigIn; 	(*Tank voll Tintenstrahldrucker Frontseite*)		(*212_A14  I3*)
	ST03_70U3_3: FB_DigIn; 	(*Fehler/Störung Tintenstrahldrucker Frontseite*)	(*212_A14  I4*)
	ST03_71U3_1: FB_DigIn; 	(*Bereit/ Im Druck Tintenstrahldrucker Rückseite*)	(*212_A14  I5*)
	ST03_71U3_2: FB_DigIn; 	(*Tank voll Tintenstrahldrucker Rückseite*)		(*212_A14  I6*)
	ST03_71U3_3: FB_DigIn; 	(*Fehler/Störung Tintenstrahldrucker Rückseite*)	(*212_A14  I7*)


	ST03_8_80_A1:FB_Sensopart;			(*Sensopart Kamera links*)			(*212_A14  I8-11*) 		(*252_A23 O3-5*)
	ST03_8_85_A1:FB_Sensopart;			(*Sensopart Kamera rechts*)		(*212_A14  I12-15*) 	(*252_A23 O6-8*)

	ST03_8_90_A1:FB_SensopartEthernet;	(*Sensopart Kamera Ethernet links*)	(*212_A14  I8-11*) 		(*252_A23 O3-5*)
	ST03_8_95_A1:FB_SensopartEthernet;	(*Sensopart Kamera Ethernet rechts*)	(*212_A14  I12-15*) 	(*252_A23 O6-8*)

	ST03_PLAN_70V1_1:FB_DigOutIn;	(* Start  Bedrucken Tintenstrahldrucker Frontseite*)	(*252_A23 O1*)
	ST03_PLAN_71V1_2:FB_DigOutIn;	(* Start  Bedrucken Tintenstrahldrucker Rückseite*) 	(*252_A23 O2*)

	ST03_Y01:FB_Valve; 				(*1: Einschaltventil Hauptluft Tintenstrahlrucker nur bei SG-Maschine 3621*)
	ST03_S18:FB_DigIn; 				(* ST02 Druckschalter Wartungseinheit Hauptluft Tintenstrahldrucker min.6 bar *)
	ST03_H6: FB_DigOutIn;			(* Signalsäule GR Bedruckubg IO *)
	ST03_H7: FB_DigOutIn;			(* Signalsäule RD Sammelstörung Bedruckung *)

(*Rüstsatz 206 pol======================================================================================*)
	ST03_435_B67_0: FB_ValveSensor; (* Förderbandeinheit  Zuführung Vereinzler AST*)
	ST03_435_B67_1: FB_ValveSensor; (* Förderbandeinheit  Zuführung Vereinzler GST*)
	ST03_435_B67_2: FB_ValveSensor; (* Förderbandeinheit  Zuführung Stopper AST*)
	ST03_435_B67_3: FB_ValveSensor; (* Förderbandeinheit  Zuführung Stopper GST*)
	ST03_435_B67_4: FB_DigIn;		(* Zuführung  frei zum Ablegen ISK SP Maschine Pos.1 *)
(*	ST03_435_B67_5: FB_DigIn;		(* Zuführung  frei zum Ablegen ISK SP Maschine Pos.2 *)
	ST03_435_B67_6: FB_DigIn;		(* Zuführung  frei zum Ablegen ISK SP Maschine Pos.3 *)*)
	ST03_435_B67_7: FB_DigIn;		(* ISK anwesend am Vereinzler*)

	ST03_436_B68_1: FB_DigIn;		(* Züführung  ISK auf Übergabeposition Roboter Palettierer Lageerkennung 1*)
	ST03_436_B68_2: FB_DigIn;		(* Züführung  ISK auf Übergabeposition Roboter Palettierer Lageerkennung 2*)
	ST03_437_B68_3: FB_DigIn;		(* Züführung  ISK auf Übergabeposition Roboter Palettierer Sender*)
	ST03_437_B68_4: FB_DigIn;		(* Züführung  ISK auf Übergabeposition Roboter Palettierer Empfänger*)
	ST03_437_Y68_5 : FB_Valve; 		(* Förderband  Zuführung Vereinzler AST/GST *)
	ST03_437_Y68_6 : FB_Valve; 		(* Förderband  Züführung Stopper AST/GST *)

(*Rüstsatz 92 pol======================================================================================*)
	ST03_444_B69_0: FB_ValveSensor; (* Förderbandeinheit  Zuführung Vereinzler AST*)
	ST03_444_B69_1: FB_ValveSensor; (* Förderbandeinheit  Zuführung Vereinzler GST*)
	ST03_444_B69_2: FB_ValveSensor; (* Förderbandeinheit  Zuführung Stopper AST*)
	ST03_444_B69_3: FB_ValveSensor; (* Förderbandeinheit  Zuführung Stopper GST*)
	ST03_444_B69_4: FB_DigIn;		(* Zuführung  frei zum Ablegen ISK SP Maschine Pos.1 *)
	ST03_444_B69_7: FB_DigIn;		(* ISK anwesend am Vereinzler*)

	ST03_445_B70_1: FB_DigIn;		(* Züführung  ISK auf Übergabeposition Roboter Palettierer Lageerkennung 1*)
	ST03_445_B70_2: FB_DigIn;		(* Züführung  ISK auf Übergabeposition Roboter Palettierer Lageerkennung 2*)
	ST03_446_B70_3: FB_DigIn;		(* Züführung  ISK auf Übergabeposition Roboter Palettierer Sender*)
	ST03_446_B70_4: FB_DigIn;		(* Züführung  ISK auf Übergabeposition Roboter Palettierer Empfänger*)
	ST03_446_Y70_5 : FB_Valve; 		(* Förderband  Zuführung Vereinzler AST/GST *)
	ST03_446_Y70_6 : FB_Valve; 		(* Förderband  Züführung Stopper AST/GST *)

(*Rüstsatz 124 pol======================================================================================*)
	ST03_451_B69_0: FB_ValveSensor; (* Förderbandeinheit  Zuführung Vereinzler AST*)
	ST03_451_B69_1: FB_ValveSensor; (* Förderbandeinheit  Zuführung Vereinzler GST*)
	ST03_451_B69_2: FB_ValveSensor; (* Förderbandeinheit  Zuführung Stopper AST*)
	ST03_451_B69_3: FB_ValveSensor; (* Förderbandeinheit  Zuführung Stopper GST*)
	ST03_451_B69_4: FB_DigIn;		(* Zuführung  frei zum Ablegen ISK SP Maschine Pos.1 *)
	ST03_451_B69_7: FB_DigIn;		(* ISK anwesend am Stopper*)

	ST03_452_B70_1: FB_DigIn;		(* Züführung  ISK auf Übergabeposition Roboter Palettierer Lageerkennung 1*)
	ST03_452_B70_2: FB_DigIn;		(* Züführung  ISK auf Übergabeposition Roboter Palettierer Lageerkennung 2*)
	ST03_453_B70_3: FB_DigIn;		(* Züführung  ISK auf Übergabeposition Roboter Palettierer Sender*)
	ST03_453_B70_4: FB_DigIn;		(* Züführung  ISK auf Übergabeposition Roboter Palettierer Empfänger*)
	ST03_453_Y70_5 : FB_Valve; 		(* Förderband  Zuführung Vereinzler AST/GST *)
	ST03_453_Y70_6 : FB_Valve; 		(* Förderband  Züführung Stopper AST/GST *)

(*Rüstsatz 46 pol======================================================================================*)
	ST03_461_B69_0: FB_ValveSensor; (* Förderbandeinheit  Zuführung Vereinzler AST*)
	ST03_461_B69_1: FB_ValveSensor; (* Förderbandeinheit  Zuführung Vereinzler GST*)
	ST03_461_B69_2: FB_ValveSensor; (* Förderbandeinheit  Zuführung Stopper AST*)
	ST03_461_B69_3: FB_ValveSensor; (* Förderbandeinheit  Zuführung Stopper GST*)
	ST03_461_B69_4: FB_DigIn;		(* Zuführung  frei zum Ablegen ISK SP Maschine Pos.1 *)
	ST03_461_B69_5: FB_ValveSensor; (* Förderbandeinheit  Zuführung  Vereinzelner Wender AST*)
	ST03_461_B69_6: FB_ValveSensor; (* Förderbandeinheit  Zuführung  Vereinzelner Wender GST*)
	ST03_461_B69_7: FB_DigIn;		(* ISK anwesend am Stopper*)

	ST03_462_B70_0: FB_DigIn;		(* Förderband  ISK anwesend Wender*)
	ST03_462_B70_1: FB_DigIn;		(* Züführung  ISK auf Übergabeposition Roboter Palettierer Lageerkennung 1*)
	ST03_462_B70_2: FB_DigIn;		(* Züführung  ISK auf Übergabeposition Roboter Palettierer Lageerkennung 2*)
	ST03_463_B70_3: FB_ValveSensor;	(* Züführung  ISK Zylinder Vakuumdüsen AST*)
	ST03_463_B70_4: FB_ValveSensor;	(* Züführung  ISK Zylinder Vakuumdüsen GST*)
	ST03_463_B70_5: FB_ValveSensor;	(* Züführung  ISK Wendestation Einlauf GST*)
	ST03_463_B70_6: FB_ValveSensor;	(* Züführung  ISK Wendestation Auslauf AST*)
	ST03_463_B70_7: FB_DigIn;		(* Züführung  ISK auf Übergabeposition Roboter Palettierer *)

	ST03_464_Y71_0 : FB_Valve; 		(* Förderband  Zuführung Vereinzelner Wender AST/GST *)
	ST03_464_Y71_1 : FB_Valve; 		(* Förderband  Zuführung Zylinder Vakuumdüsen AST/GST *)
	ST03_464_Y71_2 : FB_Valve; 		(* Förderband  Zuführung Wender Einlauf / Auslauf *)
	ST03_464_Y71_3 : FB_Valve; 		(* Förderband  Zuführung Vereinzler AST/GST *)
	ST03_464_Y71_4 : FB_Valve; 		(* Förderband  Zuführung Stopper AST/GST *)
	ST03_464_Y71_5 : FB_Valve; 		(* Förderband  Vakuumdüsen EIN/AUS *)
	ST03_464_B71_6: FB_DigIn;		(* Förderband  Vakuum vorhanden *)
	ST03_464_B71_7: FB_DigIn;		(* Förderband   Staustrecke mitte voll *)

(*Rüstsatz NOX 5+6 pol======================================================================================*)
	ST03_8_105_A1	:FB_KeyenceEtherCat; (* Keyence Kamera*)

	ST03_4x2_B69_0: FB_DigIn;			(* Zuführung frei zum Ablegen ISK SP Maschine *)
	ST03_4x2_B69_1: FB_ValveSensor; 	(* Zuführung Vereinzler GST eingefahren*)
	ST03_4x2_B69_2: FB_ValveSensor; 	(* Zuführung Vereinzler AST ausgefahren*)
	ST03_4x2_B69_3: FB_ValveSensor; 	(* Zuführung Stopper AST eingefahren*)
	ST03_4x2_B69_4: FB_ValveSensor; 	(* Zuführung Stopper GST ausgefahren*)
	ST03_4x2_B69_5: FB_DigIn;			(* ISK anwesend am Stopper *)
	ST03_4x2_B69_6: FB_ValveSensor; 	(* Zuführung Stopper Übergabeposition AST eingefahren*)
	ST03_4x2_B69_7: FB_ValveSensor; 	(* Zuführung Stopper Übergabeposition GST ausgefahren*)

	ST03_4x3_B70_0: FB_DigIn;			(* ISK anwesend Übergabeposition Stopper*)
	ST03_4x3_B70_1: FB_DigIn;			(* ISK anwesend Übergabeposition*)

	ST03_4x3_Y70_5 : FB_Valve; 			(* Zuführung Vereinzler AST/GST *)
	ST03_4x3_Y70_6 : FB_Valve; 			(* Zuführung Stopper AST/GST *)
	ST03_4x3_Y70_7 : FB_Valve; 			(* Zuführung Stopper Übergabeposition AST/GST *)

(*Rüstsatz NOX 4 pol======================================================================================*)
	ST03_491_B69_0: FB_DigIn;			(* Zuführung  frei zum Ablegen ISK SP Maschine*)
	ST03_491_B69_1: FB_ValveSensor; 	(* Förderbandeinheit  Zuführung Vereinzler AST*)
	ST03_491_B69_2: FB_ValveSensor; 	(* Förderbandeinheit  Zuführung Vereinzler GST*)
	ST03_491_B69_3: FB_ValveSensor; 	(* Förderbandeinheit  Zuführung Stopper AST*)
	ST03_491_B69_4: FB_ValveSensor; 	(* Förderbandeinheit  Zuführung Stopper GST*)
	ST03_491_B69_5: FB_DigIn;			(* ISK anwesend am Stoper*)
	ST03_491_B69_7: FB_DigIn;			(* ISK auf Abholposition Robi*)

	ST03_492_Y70_0 : FB_Valve; 			(* Förderband  Zuführung Vereinzler AST/GST *)
	ST03_492_Y70_1 : FB_Valve; 			(* Förderband  Züführung Stopper AST/GST *)

(*Rüstsatz 88 pol======================================================================================*)
	ST03_501_B69_0: FB_DigIn;			(* Zuführung  frei zum Ablegen ISK SP Maschine*)
	ST03_501_B69_1: FB_ValveSensor; 	(* Förderbandeinheit  Zuführung Vereinzler AST*)
	ST03_501_B69_2: FB_ValveSensor; 	(* Förderbandeinheit  Zuführung Vereinzler GST*)
	ST03_501_B69_3: FB_ValveSensor; 	(* Förderbandeinheit  Zuführung Stopper AST*)
	ST03_501_B69_4: FB_ValveSensor; 	(* Förderbandeinheit  Zuführung Stopper GST*)
	ST03_501_B69_5: FB_DigIn;			(* ISK anwesend am Vereinzler*)
	ST03_501_B69_6: FB_DigIn;			(* ISK anwesend am Stopper*)
	ST03_501_B69_7: FB_DigIn;			(* ISK auf Abholposition Robi*)

	ST03_502_B70_0: FB_DigIn;			(*  ISK Lageerkennung*)
	ST03_502_Y70_1 : FB_Valve; 			(* Förderband  Zuführung Vereinzler AST/GST *)
	ST03_502_Y70_2 : FB_Valve; 			(* Förderband  Züführung Stopper AST/GST *)

(*Rüstsatz 88 pol AMG==================================================================================*)
	ST03_521_B69_0: FB_DigIn;			(* Zuführung  frei zum Ablegen ISK SP Maschine*)
	ST03_521_B69_1: FB_ValveSensor; 	(* Zuführung Vereinzler eingefahren GST*)
	ST03_521_B69_2: FB_ValveSensor; 	(* Zuführung Vereinzler ausgefahren AST*)
	ST03_521_B69_3: FB_ValveSensor; 	(* Zuführung Stopper eingefahren AST*)
	ST03_521_B69_4: FB_ValveSensor; 	(* Zuführung Stopper ausgefahren GST*)

	ST03_521_B69_6: FB_DigIn;		(* ISK anwesend am Stopper*)
	ST03_521_B69_7: FB_DigIn;		(* ISK Lageerkennung links*)

	ST03_522_B70_0: FB_DigIn;		(* ISK Lageerkennung rechts*)
	ST03_522_Y70_1: FB_Valve; 		(* Zuführung Vereinzler AST/GST *)
	ST03_522_Y70_2: FB_Valve; 		(* Züführung Stopper AST/GST *)


(*Rüstsatz 7 pol======================================================================================*)
	ST03_512_XG1: FB_DigIn;				(* ISK in Klemmer*)
	ST03_512_B69_1: FB_ValveSensor; 	(* ISK Klemmer 1 AST*)
	ST03_512_B69_2: FB_ValveSensor; 	(* ISK Klemmer 1 GST*)
	ST03_512_B69_3: FB_ValveSensor; 	(* ISK Klemmer 2 AST*)
	ST03_512_B69_4: FB_ValveSensor; 	(* ISK Klemmer 2 GST*)
	ST03_512_B69_5: FB_ValveSensor; 	(* ISK Klemmer schwenkern 0° AST*)
	ST03_512_B69_6: FB_ValveSensor; 	(* ISK Klemmer schwenkern 180° GST*)


	ST03_513_B70_0: FB_ValveSensor; (* Führungsschiene  Zuführung Vereinzler AST*)
	ST03_513_B70_1: FB_ValveSensor; (* Führungsschiene  Zuführung Vereinzler GST*)
	ST03_513_B70_2: FB_ValveSensor; (* Führungsschiene  Zuführung Stopper AST*)
	ST03_513_B70_3: FB_ValveSensor; (* Führungsschiene  Zuführung Stopper GST*)
	ST03_513_B70_4: FB_DigIn;		(* ISK anwesend am Stopper*)
	ST03_513_B70_5: FB_ValveSensor; (* Übergabeposition Stopper 1 AST*)
	ST03_513_B70_6: FB_ValveSensor; (* Übergabeposition Stopper 1 GST*)
	ST03_513_B70_7: FB_DigIn;		(* ISK auf Übergabeposition 1*)

	ST03_514_B71_0: FB_ValveSensor; (* Übergabeposition Stopper 2 AST*)
	ST03_514_B71_1: FB_ValveSensor; (* Übergabeposition Stopper 2 GST*)
	ST03_514_B71_2: FB_DigIn;		(* ISK auf Übergabeposition 2*)
	ST03_514_B71_3: FB_ValveSensor; (* Übergabeposition Stopper 3 AST*)
	ST03_514_B71_4: FB_ValveSensor; (* Übergabeposition Stopper 3 GST*)
	ST03_514_B71_5: FB_DigIn;		(* ISK auf Übergabeposition 3*)
	ST03_514_B71_6: FB_DigIn;		(* ISK auf Übergabeposition 4*)
	ST03_514_B71_7: FB_DigIn;		(* Führungsschiene frei zum schwenken*)

	ST03_515_Y72_0: FB_Valve; 		(* ISK Klemmer AST/GST *)
	ST03_515_Y72_1: FB_Valve; 		(* Rinne schwenkern AST/GST *)
	ST03_515_Y72_2: FB_Valve; 		(* Führungsschiene  Zuführung Vereinzler AST/GST *)
	ST03_515_Y72_3: FB_Valve; 		(* Führungsschiene  Zuführung Stopper AST/GST *)
	ST03_515_Y72_4: FB_Valve; 		(* Übergabeposition Stopper 1  AST/GST *)
	ST03_515_Y72_5: FB_Valve; 		(* Übergabeposition Stopper 2  AST/GST *)
	ST03_515_Y72_6: FB_Valve; 		(* Übergabeposition Stopper 3  AST/GST *)

(*Rüstsatz 120 pol======================================================================================*)
	ST03_531_B69_0: FB_DigIn;			(* Zuführung  frei zum Ablegen ISK SP Maschine*)
	ST03_531_B69_1: FB_ValveSensor; 	(* Zuführung Vereinzler eingefahren GST*)
	ST03_531_B69_2: FB_ValveSensor; 	(* Zuführung Vereinzler ausgefahren AST*)
	ST03_531_B69_3: FB_ValveSensor; 	(* Zuführung Stopper eingefahren AST*)
	ST03_531_B69_4: FB_ValveSensor; 	(* Zuführung Stopper ausgefahren GST*)

	ST03_531_B69_6: FB_DigIn;			(* ISK anwesend am Stopper*)
	ST03_531_B69_7: FB_DigIn;			(* ISK rechts Lageerkennung*)

	ST03_532_B70_0: FB_DigIn;			(* ISK links Lageerkennung*)
	ST03_532_Y70_1: FB_Valve; 			(* Zuführung Vereinzler AST/GST *)
	ST03_532_Y70_2: FB_Valve; 			(* Züführung Stopper AST/GST *)

(*Rüstsatz 21 pol======================================================================================*)
	ST03_536_B69_0: FB_DigIn;			(* Zuführung  frei zum Ablegen ISK SP Maschine*)
	ST03_536_B69_1: FB_ValveSensor; 	(* Zuführung Vereinzler eingefahren GST*)
	ST03_536_B69_2: FB_ValveSensor; 	(* Zuführung Vereinzler ausgefahren AST*)
	ST03_536_B69_3: FB_ValveSensor; 	(* Zuführung Stopper eingefahren AST*)
	ST03_536_B69_4: FB_ValveSensor; 	(* Zuführung Stopper ausgefahren GST*)

	ST03_536_B69_6: FB_DigIn;			(* ISK anwesend am Stopper*)
	ST03_536_B69_7: FB_DigIn;			(* ISK anwesend an Abholposition*)

	ST03_537_B70_0: FB_DigIn;			(* ISK Lageerkennung*)
	ST03_537_Y70_1: FB_Valve; 			(* Zuführung Vereinzler AST/GST *)
	ST03_537_Y70_2: FB_Valve; 			(* Züführung Stopper AST/GST *)

(*Rüstsatz 191 pol======================================================================================*)
	ST03_541_B69_0: FB_DigIn;			(* Zuführung  frei zum Ablegen ISK SP Maschine*)
	ST03_541_B69_1: FB_ValveSensor; 	(* Zuführung Vereinzler eingefahren GST*)
	ST03_541_B69_2: FB_ValveSensor; 	(* Zuführung Vereinzler ausgefahren AST*)
	ST03_541_B69_3: FB_ValveSensor; 	(* Zuführung Stopper eingefahren AST*)
	ST03_541_B69_4: FB_ValveSensor; 	(* Zuführung Stopper ausgefahren GST*)

	ST03_541_B69_6: FB_DigIn;			(* ISK anwesend am Stopper*)
	ST03_541_B69_7: FB_DigIn;			(* ISK rechts Lageerkennung *)

	ST03_542_B70_0: FB_DigIn;			(* ISK links Lageerkennung *)
	ST03_542_Y70_1: FB_Valve; 			(* Zuführung Vereinzler AST/GST *)
	ST03_542_Y70_2: FB_Valve; 			(* Züführung Stopper AST/GST *)

(*Rüstsatz 72 pol======================================================================================*)
	ST03_546_B69_0: FB_DigIn;			(* Zuführung  frei zum Ablegen ISK SP Maschine*)
	ST03_546_B69_1: FB_ValveSensor; 	(* Zuführung Vereinzler eingefahren GST*)
	ST03_546_B69_2: FB_ValveSensor; 	(* Zuführung Vereinzler ausgefahren AST*)
	ST03_546_B69_3: FB_ValveSensor; 	(* Zuführung Stopper eingefahren AST*)
	ST03_546_B69_4: FB_ValveSensor; 	(* Zuführung Stopper ausgefahren GST*)

	ST03_546_B69_6: FB_DigIn;			(* ISK anwesend am Stopper*)
	ST03_546_B69_7: FB_DigIn;			(* ISK rechts Lageerkennung *)

	ST03_547_B70_0: FB_DigIn;			(* ISK links Lageerkennung *)
	ST03_547_Y70_1: FB_Valve; 			(* Zuführung Vereinzler AST/GST *)
	ST03_547_Y70_2: FB_Valve; 			(* Züführung Stopper AST/GST *)

(*Rüstsatz 48 pol======================================================================================*)
	ST03_551_B69_0: FB_DigIn;			(* Zuführung  frei zum Ablegen ISK SP Maschine*)
	ST03_551_B69_1: FB_ValveSensor; 	(* Zuführung Vereinzler eingefahren GST*)
	ST03_551_B69_2: FB_ValveSensor; 	(* Zuführung Vereinzler ausgefahren AST*)
	ST03_551_B69_3: FB_ValveSensor; 	(* Zuführung Stopper eingefahren AST*)
	ST03_551_B69_4: FB_ValveSensor; 	(* Zuführung Stopper ausgefahren GST*)

	ST03_551_B69_6: FB_DigIn;			(* ISK anwesend am Stopper*)
	ST03_551_B69_7: FB_DigIn;			(* ISK rechts Lageerkennung *)

	ST03_552_B70_0: FB_DigIn;			(* ISK links Lageerkennung *)
	ST03_552_Y70_1: FB_Valve; 			(* Zuführung Vereinzler AST/GST *)
	ST03_552_Y70_2: FB_Valve; 			(* Züführung Stopper AST/GST *)

(*Rüstsatz 268pol, 102pol neu======================================================================================*)

	ST03_556_B69_0	: FB_DigIn;			(* Zuführung  frei zum Ablegen ISK SP Maschine*)
	ST03_556_B69_1	: FB_ValveSensor; 	(* Zuführung Vereinzler eingefahren GST*)
	ST03_556_B69_2	: FB_ValveSensor; 	(* Zuführung Vereinzler ausgefahren AST*)
	ST03_556_B69_3	: FB_ValveSensor; 	(* Zuführung Stopper eingefahren AST*)
	ST03_556_B69_4	: FB_ValveSensor; 	(* Zuführung Stopper ausgefahren GST*)
	ST03_556_B69_5	: FB_DigIn;			(* Führungsschiene Überwachung Staustrecke*)
	ST03_556_B69_6	: FB_DigIn;			(* ISK anwesend am Stopper*)
	ST03_556_B69_7	: FB_DigIn;			(* ISK anwesend an Abholposition*)

	ST03_557_Y70_1	: FB_Valve; 		(* Zuführung Vereinzler AST/GST *)
	ST03_557_Y70_2	: FB_Valve; 		(* Züführung Stopper AST/GST *)

(*Rüstsatz 268 pol Rasterplatte======================================================================================*)
	ST03_562_B69_0: FB_DigIn;			(* Zuführung 1 frei zum schwenken*)
	ST03_562_B69_1: FB_ValveSensor; 	(* Zuführung 1 Zuführung Vereinzler GST*)
	ST03_562_B69_2: FB_ValveSensor; 	(* Zuführung 1 Zuführung Vereinzler AST*)
	ST03_562_B69_3: FB_ValveSensor; 	(* Zuführung 1 Zuführung Stopper AST*)
	ST03_562_B69_4: FB_ValveSensor; 	(* Zuführung 1 Zuführung Stopper GST*)
	(*Reserve*)
	ST03_562_B69_6: FB_DigIn;			(* Zuführung 1 ISK anwesend am Stopper*)
	ST03_562_B67_7: FB_DigIn;			(* Zuführung 1 ISK auf Übergabepos. Robi*)

	ST03_563_B70_0: FB_DigIn;			(* Zuführung 2 frei zum schwenken*)
	ST03_563_B70_1: FB_ValveSensor; 	(* Zuführung 2 Zuführung Vereinzler GST*)
	ST03_563_B70_2: FB_ValveSensor; 	(* Zuführung 2 Zuführung Vereinzler AST*)
	ST03_563_B70_3: FB_ValveSensor; 	(* Zuführung 2 Zuführung Stopper AST*)
	ST03_563_B70_4: FB_ValveSensor; 	(* Zuführung 2 Zuführung Stopper GST*)
	(*Reserve*)
	ST03_563_B70_6: FB_DigIn;			(* Zuführung 2 ISK anwesend am Stopper*)
	ST03_563_B70_7: FB_DigIn;			(* Zuführung 2 ISK auf Übergabepos. Robi*)

	ST03_564_Y71_0: FB_Valve; 			(* Zuführung 1 Vereinzler AST/GST *)
	ST03_564_Y71_1: FB_Valve; 			(* Zuführung 1 Stopper AST/GST *)
	ST03_564_Y71_2: FB_Valve; 			(* Zuführung 2 Vereinzler AST/GST *)
	ST03_564_Y71_3: FB_Valve; 			(* Zuführung 2 Stopper AST/GST *)
	ST03_564_Y71_4: FB_Valve; 			(* ISK Klemmer AST/GST *)
	ST03_564_Y71_5: FB_Valve; 			(* Rinne schwenkern AST/GST *)
	(*Reserve*)
	(*Reserve*)

	ST03_565_B72_0: FB_DigIn;			(* ISK 1 in Klemmer*)
	ST03_565_B72_1: FB_DigIn;			(* ISK 2 in Klemmer*)
	ST03_565_B72_2: FB_ValveSensor; 	(* ISK Klemmer 1 offen GST*)
	ST03_565_B72_3: FB_ValveSensor; 	(* ISK Klemmer 1 zu AST*)
	ST03_565_B72_4: FB_ValveSensor; 	(* ISK Klemmer 2 offen GST*)
	ST03_565_B72_5: FB_ValveSensor; 	(* ISK Klemmer 2 zu AST*)
	ST03_565_B72_6: FB_ValveSensor; 	(* ISK Klemmer schwenkern 0° AST*)
	ST03_565_B72_7: FB_ValveSensor; 	(* ISK Klemmer schwenkern 180° GST*)

(*Rüstsatz 33 pol======================================================================================*)

	ST03_571_B69_0	: FB_DigIn;			(* Zuführung  Pos 1 frei zum Ablegen ISK SP Maschine*)
	ST03_571_B69_1	: FB_DigIn;			(* Zuführung  Pos 2 frei zum Ablegen ISK SP Maschine*)
	ST03_571_B69_2	: FB_ValveSensor; 	(* Zuführung Vereinzler eingefahren GST*)
	ST03_571_B69_3	: FB_ValveSensor; 	(* Zuführung Vereinzler ausgefahren AST*)
	ST03_571_B69_4	: FB_ValveSensor; 	(* Zuführung Stopper eingefahren AST*)
	ST03_571_B69_5	: FB_ValveSensor; 	(* Zuführung Stopper ausgefahren GST*)
	ST03_571_B69_6	: FB_DigIn;			(* ISK anwesend am Stopper*)
	ST03_571_B69_7	: FB_DigIn;			(* ISK anwesend an Abholposition*)

	ST03_572_Y70_0	: FB_Valve; 		(* Zuführung Vereinzler AST/GST *)
	ST03_572_Y70_1	: FB_Valve; 		(* Züführung Stopper AST/GST *)

END_VAR

(* Global variable list: Station03/ST03_Global *)
VAR_GLOBAL
	gManSwivelOnRobot01		AT %QX7.2 : BOOL;
	gManSwivelOffRobot01	AT %QX7.3 : BOOL;

	Side_1            		:BOOL;
	Side_2             		:BOOL;
	gTakeTestParts 			:BOOL;
	gTakeTestPartsAuto		:BOOL;
	gTakeTestPartsFinished	:BOOL;
	NokCounter1li			:INT;
	NokCounter1re			:INT;
	NokCounter2li			:INT;
	NokCounter2re			:INT;
	NokCounter3li			:INT;
	NokCounter3re			:INT;
END_VAR

VAR_GLOBAL RETAIN PERSISTENT
	gRob01GripState			: PartState;
	gRTState				: ARRAY[1..2] OF	DINT;
 	PosIdx					: DINT;
 	gPartsInserted			: DINT;
	gPartsTest				: DINT;
	gPartsTestVisu			: DINT;		(*nur bei CZ *)
 	gNokPartsColorCam		: DINT;
 	gNokPartsWingCam		: DINT;
	gNokPartsPrint			: DINT;
	i32_first_parts			: DINT;
	i32_total_NOK_parts		: DINT;
END_VAR

(* Global variable list: Station03/ST03_VarVonfig *)
VAR_CONFIG
	(* Station 03 *)

.Robot01.RemOutStart 					AT %QX4.0 : BOOL;
.Robot01.RemOutStop 					AT %QX4.1 : BOOL;
.Robot01.RemOutPause 					AT %QX4.2 : BOOL;
.Robot01.RemOutCont 					AT %QX4.3 : BOOL;
.Robot01.RemOutReset 					AT %QX4.4 : BOOL;
.Robot01.RemOutPowerOn 				AT %QX4.5 : BOOL;
.Robot01.RemOutPowerOff 				AT %QX4.6 : BOOL;
.Robot01.RemOutPowerHi 				AT %QX4.7 : BOOL;
.Robot01.RemOutSetToolOn  			AT %QX5.0 : BOOL;
.Robot01.RemOutSetToolOff 			AT %QX5.1 : BOOL;

.Robot01.RemInReady 					AT %IX4.0 : BOOL;
.Robot01.RemInRunning 				AT %IX4.1 : BOOL;
.Robot01.RemInPaused 					AT %IX4.2 : BOOL;
.Robot01.RemInError 					AT %IX4.3 : BOOL;
.Robot01.RemInEStopOn 				AT %IX4.4 : BOOL;
.Robot01.RemInSafeguardOn		 	AT %IX4.5 : BOOL;
.Robot01.RemInSError 					AT %IX4.6 : BOOL;
.Robot01.RemInWarning 				AT %IX4.7 : BOOL;
.Robot01.RemInTcpIP_Wait 				AT %IX5.0 : BOOL;
.Robot01.RemInAreaBit1 				AT %IX5.1 : BOOL;
.Robot01.RemInAreaBit2 				AT %IX5.2 : BOOL;
.Robot01.RemInAreaBit4 				AT %IX5.3 : BOOL;
.Robot01.RemInToolCoilA   				AT %IX5.4 : BOOL;
.Robot01.RemInToolCoilB        			AT %IX5.5 : BOOL;
.Robot01.RemInToolInitSensor   			AT %IX6.0 : BOOL;
.Robot01.RemInToolWorkSensor   		AT %IX6.1 : BOOL;

(*ST03_125_F1 Absicherung Roboter (DigIn) *)
.ST03_125_F1.BitInToCheck              	AT %IX0.1 : BOOL;

(*ST03_120_A1_A14 Roboter opt.- Tool 2 ist ein (DigIn) *)
.ST03_120_A1_A14.BitInToCheck            AT %IX5.6 : BOOL;
(*ST03_400_B12_6 Schwenkmodul AST (Roboterkopf) (DigIn) *)
.ST03_400_B12_6.BitInToCheck              AT %IX6.2 : BOOL;
(*ST03_400_B12_7 Schwenkmodul GST (Roboterkopf) (DigIn) *)
.ST03_400_B12_7.BitInToCheck              AT %IX6.3 : BOOL;
(*ST03_400_B54_7 Tray Testteile in Position (DigIn) *)
.ST03_400_B54_7.BitInToCheck             AT %IX54.7 : BOOL;
(*ST03_8_75_B13_5 voll/belegt keine Prüfmittel mehr*)
.ST03_8_75_B13_5.BitInToCheck             AT %IX6.4 : BOOL;
(*ST03_8_75_B13_6 /belegt mit 6 Prüfmittel *)
.ST03_8_75_B13_6.BitInToCheck             AT %IX6.5 : BOOL;

(*Start Band für Dummyprüfung*)
.ST03_BG3_S53_0.BitInToCheck                AT %IX7.0 : BOOL;
(*LED TasterStart Band für Dummyprüfung*)
.ST03_BG3_X53_0.BitOutToSet                 AT %QX7.1 : BOOL;

(*ST03_A5 Motor Förderband Isokörper (DigOutIn) *)
.ST03_A5.BitInToCheck                : BOOL := FALSE;
.ST03_A5.BitOutToSet                 AT %QX5.2 : BOOL;

(*ST03_V2 Störung Motor Förderband (DigIn) *)
.ST03_V2.BitInToCheck              	AT %IX6.6 : BOOL;

(* Signalsäule GR Bedruckung IO *)
.ST03_H6.BitInToCheck             	: BOOL := FALSE;
.ST03_H6.BitOutToSet              	  AT %QX5.4 : BOOL;

(* Signalsäule RD Sammelstörung Bedruckung *)
.ST03_H7.BitInToCheck             	: BOOL := FALSE;
.ST03_H7.BitOutToSet              	  AT %QX5.5 : BOOL;

END_VAR

(* Global variable list: Station08/ST08_FBs *)
VAR_GLOBAL

	ST08_400_B50_0 : FB_DigIn; (* Traystapel vor Vereinzeler Einlaufband hinten *)
	ST08_400_B50_4 : FB_ValveSensor; (* Stopper Traystapel Einlaufband hinten rechts GST *)
	ST08_401_B50_5 : FB_DigIn; (* Traystapel vor Vereinzeler Einlaufband mitte *)
	ST08_401_B50_7 : FB_ValveSensor; (* Traystapel schieben hinten ausgefahren *)
	ST08_401_B51_1 : FB_ValveSensor; (* Stopper Traystapel Einlaufband mitte rechts GST *)
	ST08_402_B51_2 : FB_DigIn; (* Traystapel vor Vereinzeler Einlaufband vorne *)
	ST08_402_B51_3 : FB_ValveSensor; (* Traystapel schieben mitte ausgefahren *)
	ST08_402_B51_6 : FB_ValveSensor; (* Stopper Traystapel Einlaufband vorne rechts GST *)
	ST08_402_B51_4 : FB_DigIn; (* Luftzone 1 *)
	ST08_402_B51_5 : FB_DigIn; (* Luftzone 2 *)
	ST08_402_B51_7 : FB_ValveSensor; (* Traystapel schieben vorne ausgefahren *)

	ST08_403_B52_0 : FB_ValveSensor; (* Hubtüre 1 Einlauf STN8 AST *)
	ST08_403_B52_1 : FB_ValveSensor; (* Hubtüre 1 Einlauf STN8 GST *)
	ST08_404_B52_2 : FB_DigIn; (* Traystapel in Ablageposition Isokörper *)
	ST08_404_B52_3 : FB_DigIn; (* Traystapel richtig eingelegt Isokörper *)
	ST08_404_B52_4 : FB_ValveSensor; (* Stopper Traystapel Isokörper AST *)
	ST08_404_B52_5 : FB_ValveSensor; (* Stopper Traystapel Isokörper GST *)
	ST08_404_B52_6 : FB_ValveSensor; (* Abstapelzylinder 1 Isokörper AST *)
	ST08_404_B52_7 : FB_ValveSensor; (* Abstapelzylinder 1 Isokörper GST *)
	ST08_404_B53_0 : FB_ValveSensor; (* Abstapelzylinder 2 Isokörper AST *)
	ST08_404_B53_1 : FB_ValveSensor; (* Abstapelzylinder 2 Isokörper GST *)
	ST08_405_B53_2 : FB_ValveSensor; (* Rückhaltezylinder links Traystapel Isokörper AST *)
	ST08_405_B53_3 : FB_ValveSensor; (* Rückhaltezylinder links Traystapel Isokörper GST *)
	ST08_405_B53_4 : FB_ValveSensor; (* Rückhaltezylinder rechts Traystapel Isokörper AST *)
	ST08_405_B53_5 : FB_ValveSensor; (* Rückhaltezylinder rechts Traystapel Isokörper GST *)
	ST08_405_B53_6 : FB_ValveSensor; (* Hubtüre 2 Einlauf Isokörper STN8 AST *)
	ST08_405_B53_7 : FB_ValveSensor; (* Hubtüre 2 Einlauf Isokörper STN8 GST *)
	ST08_406_B54_0 : FB_DigIn; (* Tray in Zwischenp. Entnahme Isokörper (Bandende) *)
	ST08_406_B54_1 : FB_ValveSensor; (* Hub Bandstrecke 2und 3 STN8 AST *)
	ST08_406_B54_2 : FB_ValveSensor; (* Hub Bandstrecke 2und 3 STN8 GST *)
	ST08_406_B54_3 : FB_DigIn; (* Ausheber Trays in Entnahmepos *)
	ST08_406_B54_4 : FB_ValveSensor; (* Ausheber Trays Entnahmepos. Isok. STN8 AST *)
	ST08_406_B54_5 : FB_ValveSensor; (* Ausheber Trays Entnahmepos. Isok. STN8 GST *)
	ST08_406_B54_6 : FB_DigIn; (* Tray aus Entnahme ausgelaufen (Bandende) *)
	ST08_407_B55_0 : FB_ValveSensor; (* Hubtüre 3 Auslauf STN8 AST *)
	ST08_407_B55_1 : FB_ValveSensor; (* Hubtüre 3 Auslauf STN8 GST *)
	ST08_407_B55_2 : FB_ValveSensor; (* Hubtüre 4 Auslauf STN8 AST *)
	ST08_407_B55_3 : FB_ValveSensor; (* Hubtüre 4 Auslauf STN8 GST *)
	ST08_407_B55_4 : FB_DigIn; (* Tray in Aufstapelposition eingelaufen STN8 *)
	ST08_409_B55_5 : FB_DigIn; (* Auslaufrollenbahn voll STN8 *)

	ST08_408_B56_0 : FB_ValveSensor; (* Rückhaltezylinder links Auslauf STN8 AST *)
	ST08_408_B56_1 : FB_ValveSensor; (* Rückhaltezylinder links Auslauf STN8 GST *)
	ST08_408_B56_2 : FB_ValveSensor; (* Rückhaltezylinder rechts Auslauf STN8 AST *)
	ST08_408_B56_3 : FB_ValveSensor; (* Rückhaltezylinder rechts Auslauf STN8 GST *)
	ST08_408_B56_4 : FB_ValveSensor; (* Abstapelzylinder 1 STN8 AST *)
	ST08_408_B56_5 : FB_ValveSensor; (* Abstapelzylinder 1 STN8 GST *)
	ST08_408_B56_6 : FB_ValveSensor; (* Abstapelzylinder 2 STN8 AST *)
	ST08_408_B56_7 : FB_ValveSensor; (* Abstapelzylinder 2 STN8 AST *)

	ST08_400_B50_1: FB_ValveSensor; (* Stopper links + rechts Traystapel Auslaufband eingefahren*)
	ST08_400_B50_2: FB_ValveSensor; (* Stopper links + rechts Traystapel Auslaufband ausgefahren*)
	ST08_400_B50_3: FB_ValveSensor; (* Stopper links + rechts Traystapel Auslaufband eingefahren*)
	ST08_400_B50_6: FB_ValveSensor; (* Stopper links + rechts Traystapel Auslaufband ausgefahren*)

	(*Rüstsatz 74, 91, 168,35 pol*)
	ST08_412_B58_0: FB_ValveSensor; 	(* Rüstsatz Förderband Vereinzelner eingefahren*)
	ST08_412_B58_1: FB_ValveSensor; 	(* Rüstsatz Förderband Vereinzelner ausgefahren*)
	ST08_412_B58_2: FB_ValveSensor; 	(* Rüstsatz Förderband Stopper eingefahren*)
	ST08_412_B58_3: FB_ValveSensor; 	(* Rüstsatz Förderband Stopper ausgefahren*)
	ST08_412_B58_4: FB_DigIn;		(*  Rüstsatz Förderband frei zum Ablegen ISK von SP Maschine Position 1 *)		(*35pol ISK zum Ablegen  frei für SP Maschine*)
	ST08_412_B58_5: FB_DigIn;		(*  Rüstsatz Förderband frei zum Ablegen ISK von SP Maschine Position 2 *)
	ST08_412_B58_6: FB_DigIn;		(*  Rüstsatz Förderband frei zum Ablegen ISK von SP Maschine Position 3 *)
	ST08_412_B58_5_35pol: FB_DigIn;	(*35pol Lageerkennung links*)
	ST08_412_B58_6_35pol: FB_DigIn;	(*35pol Lageerkennung rechts*)
	ST08_412_B58_7: FB_DigIn;		(*  Rüstsatz Förderband ISK anwesend zum Vereinzeln *)
	ST08_412_B59_0: FB_DigIn;		(*  Rüstsatz Förderband ISK auf Übergabeposition Roboter Verpackung *)

	ST08_412_Y55_0 : FB_Valve; (* Rüstsatz Förderband Vereinzelner einfahren *)
	ST08_412_Y55_2 : FB_Valve; (* Rüstsatz Förderband Stopper einfahren *)

	(*=================*)

	ST08_169_K1 : FB_DigOutIn; (* Bandantrieb 1 Einlauf Trays Ein *)
	ST08_169_K2 : FB_DigOutIn; (* Bandantrieb 4 Auslauf leere Trays Ein *)
	ST08_170_K1 : FB_DigOutIn; (* Bandantrieb 2 Hubquereinheit Trays Ein *)
	ST08_170_K2 : FB_DigOutIn; (* Bandantrieb 3 Hubquereinheit Trays Ein *)

	ST08_400_Y50_0 : FB_Valve; (* Stopper Traystapel Einlaufb. hinten links + rechts AST *)
	ST08_400_Y50_2 : FB_Valve; (* Stopper Traystapel Einlaufb. mitte links + rechts AST *)
	ST08_402_Y50_4 : FB_Valve; (* Stopper Traystapel Einlaufb. vorne links + rechts AST *)
	ST08_403_Y50_6 : FB_Valve; (* Vakuum 1 Einlauf STN8 *)
	ST08_403_Y50_7 : FB_Valve; (* Vakuum 2 Einlauf STN8 *)
	ST08_405_Y51_0 : FB_Valve; (* Hubtüre 2 Einlauf Isokörper STN8 AST *)

	ST08_404_Y51_6 : FB_Valve; (* Stopper Traystapel Isokörper AST *)

	ST08_406_Y51_2 : FB_Valve; (* Hubtüre 3 Auslauf  STN8 AST *)
	ST08_407_Y51_4 : FB_Valve; (* Hubtüre 4 Auslauf STN8 AST *)
	ST08_404_Y52_0 : FB_Valve; (* Hub Bandstrecke AST *)
	ST08_406_Y52_3 : FB_Valve; (* Ausheber Trays Entnahmepos. Isok. STN8 GST *)
	ST08_401_Y52_4 : FB_Valve; (* Traystapel schieben hinten AST*)
	ST08_400_Y52_5 : FB_Valve; (* Stopper links + rechts Traystapel Auslaufband einfahren *)
	ST08_402_Y52_6 : FB_Valve; (* Traystapel schieben mitte AST*)
	ST08_402_Y52_7 : FB_Valve; (* Traystapel schieben vorne AST *)
	ST08_404_Y53_0 : FB_Valve; (* Abstapelzylinder 1 Isokörper AST *)
	ST08_404_Y53_2 : FB_Valve; (* Abstapelzylinder 2 Isokörper AST *)

	ST08_405_Y53_4 : FB_Valve; (* Rückhaltezylinder li+re Traystapel Isokörper AST *)
	ST08_408_Y54_0 : FB_Valve; (* Rückhaltezylinder li.+re. Auslauf STN8 AST *)
	ST08_408_Y54_2 : FB_Valve; (* Abstapelzylinder 1 STN8 AST *)
	ST08_408_Y54_4 : FB_Valve; (* Abstapelzylinder 2 STN8 AST *)


	ST08_180_M1			:fb_72x1_Achse;		(*Abstapeln*)
	ST08_180_M1_ON		:fb_Auto_On_Off;	(*Abstapeln*)

	ST08_185_M1			:fb_72x1_Achse;		(*Aufstapeln*)
	ST08_185_M1_ON		:fb_Auto_On_Off;	(*Abstapeln*)

	ST08_190_M1			:fb_72x1_Achse;		(*Tray ausheben*)
	ST08_190_M1_ON		:fb_Auto_On_Off;	(*Tray ausheben*)
END_VAR

(* Global variable list: Station08/ST08_Global *)
VAR_GLOBAL

END_VAR
VAR_GLOBAL RETAIN PERSISTENT
	gRequestNewStack		:BOOL;
	gNewStackIn				:BOOL;
END_VAR

(* Global variable list: Station08/ST08_VarVonfig *)
VAR_CONFIG

(*ST08_400_B50_0 Traystapel vor Vereinzeler Einlaufband hinten (DigIn) *)
.ST08_400_B50_0.BitInToCheck             AT %IX50.0 : BOOL;
(*ST08_400_B50_1 Stopper links + rechts Traystapel Auslaufband eingefahren (DigIn) *)
.ST08_400_B50_1.ValveSensor             AT %IX50.1 : BOOL;
(*ST08_400_B50_2 Stopper links + rechts Traystapel Auslaufband ausgefahren (DigIn) *)
.ST08_400_B50_2.ValveSensor             AT %IX50.2 : BOOL;
(*ST08_400_B50_3 Stopper links + rechts Traystapel Auslaufband eingefahren (DigIn) *)
.ST08_400_B50_3.ValveSensor             AT %IX50.3 : BOOL;
(*ST08_400_B50_4 Stopper Traystapel Einlaufband hinten rechts GST (DigIn) *)
.ST08_400_B50_4.ValveSensor             AT %IX50.4 : BOOL;
(*ST08_401_B50_5 Traystapel vor Vereinzeler Einlaufband mitte (DigIn) *)
.ST08_401_B50_5.BitInToCheck             AT %IX50.5 : BOOL;
(*ST08_400_B50_6 Stopper links + rechts Traystapel Auslaufband ausgefahren (DigIn) *)
.ST08_400_B50_6.ValveSensor             AT %IX50.6 : BOOL;
(*ST08_401_B50_7 Traystapel schieben hinten ausgefahren (DigIn) *)
.ST08_401_B50_7.ValveSensor             AT %IX50.7 : BOOL;

(*ST08_401_B51_1 Stopper Traystapel Einlaufband mitte rechts GST (DigIn) *)
.ST08_401_B51_1.ValveSensor             AT %IX51.1 : BOOL;
(*ST08_402_B51_2 Traystapel vor Vereinzeler Einlaufband vorne (DigIn) *)
.ST08_402_B51_2.BitInToCheck             AT %IX51.2 : BOOL;
(*ST08_402_B51_3 Traystapel schieben mitte ausgefahren (DigIn) *)
.ST08_402_B51_3.ValveSensor             AT %IX51.3 : BOOL;
(*ST08_402_B51_4  (* Luftzone 1 *) (DigIn) *)
.ST08_402_B51_4.BitInToCheck             AT %IX51.4 : BOOL;
(*ST08_402_B51_5  (* Luftzone 2 *) (DigIn) *)
.ST08_402_B51_5.BitInToCheck             AT %IX51.5 : BOOL;
(*ST08_402_B51_6 Stopper Traystapel Einlaufband vorne rechts GST (DigIn) *)
.ST08_402_B51_6.ValveSensor             AT %IX51.6 : BOOL;
(*ST08_402_B51_7 Traystapel schieben vorne ausgefahren (DigIn) *)
.ST08_402_B51_7.ValveSensor             AT %IX51.7 : BOOL;

(*ST08_403_B52_0 Hubtüre 1 Einlauf STN8 AST (DigIn) *)
.ST08_403_B52_0.ValveSensor             AT %IX52.0 : BOOL;
(*ST08_403_B52_1 Hubtüre 1 Einlauf STN8 GST (DigIn) *)
.ST08_403_B52_1.ValveSensor             AT %IX52.1 : BOOL;
(*ST08_404_B52_2 Traystapel in Ablageposition Isokörper (DigIn) *)
.ST08_404_B52_2.BitInToCheck             AT %IX52.2 : BOOL;
(*ST08_404_B52_3 Traystapel richtig eingelegt Isokörper (DigIn) *)
.ST08_404_B52_3.BitInToCheck             AT %IX52.3 : BOOL;
(*ST08_404_B52_4 Stopper Traystapel Isokörper AST (DigIn) *)
.ST08_404_B52_4.ValveSensor             AT %IX52.4 : BOOL;
(*ST08_404_B52_5 Stopper Traystapel Isokörper GST (DigIn) *) 
.ST08_404_B52_5.ValveSensor             AT %IX52.5 : BOOL;
(*ST08_404_B52_6 Abstapelzylinder 1 Isokörper AST (DigIn) *) 
.ST08_404_B52_6.ValveSensor             AT %IX52.6 : BOOL;
(*ST08_404_B52_7 Abstapelzylinder 1 Isokörper GST (DigIn) *) 
.ST08_404_B52_7.ValveSensor             AT %IX52.7 : BOOL;
(*ST08_404_B53_0 Abstapelzylinder 2 Isokörper AST (DigIn) *)
.ST08_404_B53_0.ValveSensor             AT %IX53.0 : BOOL;
(*ST08_404_B53_1 Abstapelzylinder 2 Isokörper GST (DigIn) *)
.ST08_404_B53_1.ValveSensor             AT %IX53.1 : BOOL;
(*ST08_405_B53_2 Rückhaltezylinder links Traystapel Isokörper AST (DigIn) *) 
.ST08_405_B53_2.ValveSensor             AT %IX53.2 : BOOL;
(*ST08_405_B53_3 Rückhaltezylinder links Traystapel Isokörper GST (DigIn) *) 
.ST08_405_B53_3.ValveSensor             AT %IX53.3 : BOOL;
(*ST08_405_B53_4 Rückhaltezylinder rechts Traystapel Isokörper AST (DigIn) *) 
.ST08_405_B53_4.ValveSensor             AT %IX53.4 : BOOL;
(*ST08_405_B53_5 Rückhaltezylinder rechts Traystapel Isokörper GST (DigIn) *)
.ST08_405_B53_5.ValveSensor             AT %IX53.5 : BOOL;
(*ST08_405_B53_6 Hubtüre 2 Einlauf Isokörper STN8 AST (DigIn) *)
.ST08_405_B53_6.ValveSensor             AT %IX53.6 : BOOL;
(*ST08_405_B53_7 Hubtüre 2 Einlauf Isokörper STN8 GST (DigIn) *)
.ST08_405_B53_7.ValveSensor             AT %IX53.7 : BOOL;
(*ST08_406_B54_0 Tray in Zwischenp. Entnahme Isokörper (Bandende) (DigIn) *)
.ST08_406_B54_0.BitInToCheck             AT %IX54.0 : BOOL;
(*ST08_406_B54_1 Hub Bandstrecke 2und 3 STN8 AST (DigIn) *)
.ST08_406_B54_1.ValveSensor             AT %IX54.1 : BOOL;
(*ST08_406_B54_2 Hub Bandstrecke 2und 3 STN8 GST (DigIn) *) 
.ST08_406_B54_2.ValveSensor             AT %IX54.2 : BOOL;
(*ST08_406_B54_3  Traystapel in Ausheber Isokörper GST (DigIn) *)
.ST08_406_B54_3.BitInToCheck             AT %IX54.3 : BOOL;
(*ST08_406_B54_4 Ausheber Trays Entnahmepos. Isok. STN8 AST (DigIn) *)
.ST08_406_B54_4.ValveSensor             AT %IX54.4 : BOOL;
(*ST08_406_B54_5 Ausheber Trays Entnahmepos. Isok. STN8 GST (DigIn) *)
.ST08_406_B54_5.ValveSensor             AT %IX54.5 : BOOL;
(*ST08_406_B54_6 Tray aus Entnahme Isokörper (Bandende) (DigIn) *)
.ST08_406_B54_6.BitInToCheck             AT %IX54.6 : BOOL;
(*ST08_407_B55_0 Hubtüre 3 Auslauf STN8 AST (DigIn) *)
.ST08_407_B55_0.ValveSensor             AT %IX55.0 : BOOL;
(*ST08_407_B55_1 Hubtüre 3 Auslauf STN8 GST (DigIn) *)
.ST08_407_B55_1.ValveSensor             AT %IX55.1 : BOOL;
(*ST08_407_B55_2 Hubtüre 4 Auslauf STN8 AST (DigIn) *)
.ST08_407_B55_2.ValveSensor             AT %IX55.2 : BOOL;
(*ST08_407_B55_3 Hubtüre 4 Auslauf STN8 GST (DigIn) *)
.ST08_407_B55_3.ValveSensor             AT %IX55.3 : BOOL;
(*ST08_407_B55_4 Tray in Aufstapelposition eingelaufen STN8 (DigIn) *)
.ST08_407_B55_4.BitInToCheck             AT %IX55.4 : BOOL;
(*ST08_409_B55_5 Auslaufrollenbahn voll STN8 (DigIn) *)
.ST08_409_B55_5.BitInToCheck             AT %IX55.5 : BOOL;
(*ST08_408_B56_0 Rückhaltezylinder links Auslauf STN8 AST (DigIn) *)
.ST08_408_B56_0.ValveSensor             AT %IX56.0 : BOOL;
(*ST08_408_B56_1 Rückhaltezylinder links Auslauf STN8 GST (DigIn) *) 
.ST08_408_B56_1.ValveSensor             AT %IX56.1 : BOOL;
(*ST08_408_B56_2 Rückhaltezylinder rechts Auslauf STN8 AST (DigIn) *)
.ST08_408_B56_2.ValveSensor             AT %IX56.2 : BOOL;
(*ST08_408_B56_3 Rückhaltezylinder rechts Auslauf STN8 GST (DigIn) *) 
.ST08_408_B56_3.ValveSensor             AT %IX56.3 : BOOL;
(*ST08_408_B56_4 Abstapelzylinder 1 STN8 AST (DigIn) *)
.ST08_408_B56_4.ValveSensor             AT %IX56.4 : BOOL;
(*ST08_408_B56_5 Abstapelzylinder 1 STN8 GST (DigIn) *) 
.ST08_408_B56_5.ValveSensor             AT %IX56.5 : BOOL;
(*ST08_408_B56_6 Abstapelzylinder 2 STN8 AST (DigIn) *) 
.ST08_408_B56_6.ValveSensor             AT %IX56.6 : BOOL;
(*ST08_408_B56_7 Abstapelzylinder 2 STN8 AST (DigIn) *) 
.ST08_408_B56_7.ValveSensor             AT %IX56.7 : BOOL;

(*ST08_412_B58_0 Rüstsatz Förderband Vereinzelner eingefahren (DigIn) *)
.ST08_412_B58_0.ValveSensor             AT %IX58.0 : BOOL;
(*ST08_412_B58_1 Rüstsatz Förderband Vereinzelner ausgefahren (DigIn) *)
.ST08_412_B58_1.ValveSensor             AT %IX58.1 : BOOL;
(*ST08_412_B58_2 Rüstsatz Förderband Stopper eingefahren (DigIn) *)
.ST08_412_B58_2.ValveSensor             AT %IX58.2 : BOOL;
(*ST08_412_B58_3 Rüstsatz Förderband Stopper ausgefahren (DigIn) *)
.ST08_412_B58_3.ValveSensor             AT %IX58.3 : BOOL;
(*ST08_412_B58_4 Rüstsatz Förderband frei zum Ablegen ISK von SP Maschine Position 1 (DigIn) *)
.ST08_412_B58_4.BitInToCheck             AT %IX58.4 : BOOL;
(*ST08_412_B58_5 Rüstsatz Förderband frei zum Ablegen ISK von SP Maschine Position 2 (DigIn) *)
.ST08_412_B58_5.BitInToCheck             AT %IX58.5 : BOOL;
(*ST08_412_B58_6 Rüstsatz Förderband frei zum Ablegen ISK von SP Maschine Position 3 (DigIn) *)
.ST08_412_B58_6.BitInToCheck             AT %IX58.6 : BOOL;
(*(*ST08_412_B58_5_35pol Lagerekennung links (DigIn) *)
.ST08_412_B58_5_35pol.BitInToCheck             AT %I* : BOOL;
(*ST08_412_B58_6_35pol Lageerkennung rechts (DigIn) *)
.ST08_412_B58_6_35pol.BitInToCheck             AT %I* : BOOL;*)

(*ST08_412_B58_7 Rüstsatz Förderband ISK anwesend zum Vereinzeln (DigIn) *)
.ST08_412_B58_7.BitInToCheck             AT %IX58.7 : BOOL;
(*ST08_412_B59_0 Rüstsatz Förderband ISK auf Übergabeposition Roboter Verpackung (DigIn) *)
.ST08_412_B59_0.BitInToCheck             AT %IX59.0 : BOOL;

(*ST08_169_K1 Bandantrieb 1 Einlauf Trays Ein (DigOutIn) *)
.ST08_169_K1.BitInToCheck                : BOOL := FALSE;
.ST08_169_K1.BitOutToSet                 AT %QX3.3 : BOOL;
(*ST08_169_K2 Bandantrieb 4 Auslauf leere Trays Ein (DigOutIn) *)
.ST08_169_K2.BitInToCheck                : BOOL := FALSE;
.ST08_169_K2.BitOutToSet                 AT %QX3.4 : BOOL;
(*ST08_170_K1 Bandantrieb 2 Hubquereinheit Trays Ein (DigOutIn) *)
.ST08_170_K1.BitInToCheck                : BOOL := FALSE;
.ST08_170_K1.BitOutToSet                 AT %QX3.5 : BOOL;
(*ST08_170_K2 Bandantrieb 3 Hubquereinheit Trays Ein (DigOutIn) *)
.ST08_170_K2.BitInToCheck                : BOOL := FALSE;
.ST08_170_K2.BitOutToSet                 AT %QX3.6 : BOOL;
(*ST08_400_Y50_0 Stopper Traystapel Einlaufb. hinten links + rechts AST (Valve) *)
.ST08_400_Y50_0.CoilA                    AT %QX50.0 : BOOL;
.ST08_400_Y50_0.CoilB                    AT %QX50.1 : BOOL;
(*ST08_400_Y50_2 Stopper Traystapel Einlaufb. mitte links + rechts AST (Valve) *)
.ST08_400_Y50_2.CoilA                    AT %QX50.2 : BOOL;
.ST08_400_Y50_2.CoilB                    AT %QX50.3 : BOOL;
(*ST08_402_Y50_4 Stopper Traystapel Einlaufb. vorne links + rechts AST (Valve) *) 
.ST08_402_Y50_4.CoilA                    AT %QX50.4 : BOOL;
.ST08_402_Y50_4.CoilB                    AT %QX50.5 : BOOL;
(*ST08_403_Y50_6 Vakuum 1 Einlauf STN8 AST (Valve) *)
.ST08_403_Y50_6.CoilA                    AT %QX50.6 : BOOL;
.ST08_403_Y50_6.CoilB                    AT %MX50.6 : BOOL;
(*ST08_403_Y50_7 Vakuum 2 Einlauf STN8 AST (Valve) *)
.ST08_403_Y50_7.CoilA                    AT %QX50.7 : BOOL;
.ST08_403_Y50_7.CoilB                    AT %MX50.7 : BOOL;
(*ST08_405_Y51_0 Hubtüre 2 Einlauf Isokörper STN8 AST (Valve) *)
.ST08_405_Y51_0.CoilA                    AT %QX51.0 : BOOL;
.ST08_405_Y51_0.CoilB                    AT %QX51.1 : BOOL;
(*ST08_406_Y51_2 Hubtüre 3 STN8 AST (Valve) *)
.ST08_406_Y51_2.CoilA                    AT %QX51.2 : BOOL;
.ST08_406_Y51_2.CoilB                    AT %QX51.3 : BOOL;
(*ST08_407_Y51_4 Hubtüre 4 Auslauf STN8 AST (Valve) *)
.ST08_407_Y51_4.CoilA                    AT %QX51.4 : BOOL;
.ST08_407_Y51_4.CoilB                    AT %QX51.5 : BOOL;
(*ST08_404_Y51_6 Stopper Traystapel Isokörper AST (Valve) *)
.ST08_404_Y51_6.CoilA                    AT %QX51.6 : BOOL;
.ST08_404_Y51_6.CoilB                    AT %QX51.7 : BOOL;

(*ST08_404_Y52_0 Hub Bandstrecke STN8 AST (Valve) *)
.ST08_404_Y52_0.CoilA                    AT %QX52.0 : BOOL;
.ST08_404_Y52_0.CoilB                    AT %QX52.1 : BOOL;
(*ST08_406_Y52_3 Ausheber Trays Entnahmepos. Isok. STN8 GST (Valve) *)
.ST08_406_Y52_3.CoilA                    AT %QX52.2 : BOOL;
.ST08_406_Y52_3.CoilB                    AT %QX52.3 : BOOL;
	(* Traystapel schieben hinten ausfahren (Valve) *)
	.ST08_401_Y52_4.CoilA                    AT %QX52.4 : BOOL;
	.ST08_401_Y52_4.CoilB                    AT %MX52.4 : BOOL;
(* Stopper links + rechts Traystapel Auslaufband einfahren (Valve) *)
.ST08_400_Y52_5.CoilA                    AT %QX52.5 : BOOL;
.ST08_400_Y52_5.CoilB                    AT %MX52.5 : BOOL;
	(* Traystapel schieben mitte ausfahren (Valve) *)
	.ST08_402_Y52_6.CoilA                    AT %QX52.6 : BOOL;
	.ST08_402_Y52_6.CoilB                    AT %MX52.6 : BOOL;
	(* Traystapel schieben mitte ausfahren (Valve) *)
	.ST08_402_Y52_7.CoilA                   AT %QX52.7 : BOOL;
	.ST08_402_Y52_7.CoilB                    AT %MX52.7 : BOOL;
(*ST08_404_Y53_0 Abstapelzylinder 1 Isokörper AST (Valve) *)
.ST08_404_Y53_0.CoilA                    AT %QX53.0 : BOOL;
.ST08_404_Y53_0.CoilB                    AT %QX53.1 : BOOL;
(*ST08_404_Y53_2 Abstapelzylinder 2 Isokörper AST (Valve) *)
.ST08_404_Y53_2.CoilA                    AT %QX53.2 : BOOL;
.ST08_404_Y53_2.CoilB                    AT %QX53.3 : BOOL;
(*ST08_405_Y53_4 Rückhaltezylinder li+re Traystapel Isokörper AST (Valve) *)
.ST08_405_Y53_4.CoilA                    AT %QX53.4 : BOOL;
.ST08_405_Y53_4.CoilB                    AT %QX53.5 : BOOL;
(*ST08_408_Y54_0 Rückhaltezylinder li.+re. Auslauf STN8 AST (Valve) *)
.ST08_408_Y54_0.CoilA                    AT %QX54.0 : BOOL;
.ST08_408_Y54_0.CoilB                    AT %QX54.1 : BOOL;
(*ST08_408_Y54_2 Abstapelzylinder 1 STN8 AST (Valve) *)
.ST08_408_Y54_2.CoilA                    AT %QX54.2 : BOOL;
.ST08_408_Y54_2.CoilB                    AT %QX54.3 : BOOL;
(*ST08_408_Y54_4 Abstapelzylinder 2 STN8 AST (Valve) *)
.ST08_408_Y54_4.CoilA                    AT %QX54.4 : BOOL;
.ST08_408_Y54_4.CoilB                    AT %QX54.5 : BOOL;
(*ST08_412_Y55_0 Rüstsatz Förderband Vereinzelner (Valve) *)
.ST08_412_Y55_0.CoilA                    AT %QX55.0 : BOOL;
.ST08_412_Y55_0.CoilB                    AT %QX55.1 : BOOL;
(*ST08_412_Y55_2 Rüstsatz Förderband Stopper (Valve) *)
.ST08_412_Y55_2.CoilA                    AT %QX55.2 : BOOL;
.ST08_412_Y55_2.CoilB                    AT %QX55.3 : BOOL;

END_VAR

